// (3) per-StepNo aggregate (find-or-allocate; fixed array, Core §8.11.4(e))
slot := 0;
FOR i := 1 TO PL_Fraktal.MAX_PROFILE_STEPS DO
    IF (StepStats[i].Count > 0) AND (StepStats[i].Id = _openNo) THEN
        slot := i;
        EXIT;
    ELSIF (slot = 0) AND (StepStats[i].Count = 0) THEN
        slot := i;
    END_IF
END_FOR
IF slot = 0 THEN
    StatsTruncated := TRUE;
ELSE
    StepStats[slot].Id    := _openNo;
    StepStats[slot].Label := _openName;
    StepStats[slot].Class := _openClass;
    F_TimingUpdate(Row := StepStats[slot], DurMs := dur);
END_IF
END_METHOD

END_FUNCTION_BLOCK

// ---- BaseClasses/FB_CompositeModuleBase.TcPOU
// Core §2.2 / §8.2 — CM lifecycle + child registry + first-out rollup.
// An EM type registers its children in Setup (_M_Register), ticks them every scan
// (_M_TickChildren, so status stays live whether or not a command runs — Annex B),
// and adopts the first faulted child's diagnostic verbatim (_M_RollupFault).
{attribute 'OPC.UA.DA' := '1'}
FUNCTION_BLOCK ABSTRACT FB_CompositeModuleBase EXTENDS FB_ModuleBase
VAR
    _children : ARRAY[1..PL_Fraktal.MAX_EM_CHILDREN] OF I_Module;
    _nChild   : INT;
END_VAR

Cyclic();

// called from the type's Setup (Core §3.11); bounds-checked per Core §5.6
METHOD PROTECTED _M_Register : BOOL
VAR_INPUT
    Child : I_Module;
END_VAR
IF (Child = 0) OR (_nChild >= PL_Fraktal.MAX_EM_CHILDREN) THEN
    _M_Register := FALSE;
    RETURN;
END_IF
_nChild := _nChild + 1;
_children[_nChild] := Child;
_M_Register := TRUE;
END_METHOD

METHOD PrepareRecipe : BOOL
VAR_INPUT
    Model : ST_ModelId;
END_VAR
VAR
    i, j : INT;
END_VAR
PrepareRecipe := TRUE;
FOR i := 1 TO _nChild DO
    IF (_children[i] <> 0) AND_THEN NOT _children[i].PrepareRecipe(Model := Model) THEN
        PrepareRecipe := FALSE;
        FOR j := 1 TO i DO
            IF _children[j] <> 0 THEN _children[j].AbortRecipe(); END_IF
        END_FOR
        RETURN;
    END_IF
END_FOR
END_METHOD

METHOD CommitRecipe
VAR
    i : INT;
END_VAR
FOR i := 1 TO _nChild DO
    IF _children[i] <> 0 THEN _children[i].CommitRecipe(); END_IF
END_FOR
END_METHOD

METHOD AbortRecipe
VAR
    i : INT;
END_VAR
FOR i := 1 TO _nChild DO
    IF _children[i] <> 0 THEN _children[i].AbortRecipe(); END_IF
END_FOR
END_METHOD

// Core §8.2 — adopt the FIRST faulted child's first-out (reason + child SourcePath)
METHOD PROTECTED _M_RollupFault : BOOL
VAR
    i : INT;
END_VAR
_M_RollupFault := FALSE;
FOR i := 1 TO _nChild DO
    IF _children[i] <> 0 AND_THEN _children[i].FaultActive THEN
        _M_FaultDiag(_children[i].GetFaultSummary());
        _M_RollupFault := TRUE;
        RETURN;
    END_IF
END_FOR
END_METHOD

// children always tick so their status stays live (Annex B §B.3)
METHOD PROTECTED _M_TickChildren
VAR
    i : INT;
END_VAR
FOR i := 1 TO _nChild DO
    IF _children[i] <> 0 THEN
        _children[i].Cyclic();
    END_IF
END_FOR
END_METHOD

PROPERTY ModuleType : E_ModuleType
GET
ModuleType := E_ModuleType.NONE;
END_GET
END_PROPERTY

END_FUNCTION_BLOCK

// ---- BaseClasses/FB_EquipmentModuleBase.TcPOU
// Core §2.2 — discrete-command composite tier. Child recursion lives in
// FB_CompositeModuleBase; this type supplies Equipment Module identity/capability.
FUNCTION_BLOCK ABSTRACT FB_EquipmentModuleBase EXTENDS FB_CompositeModuleBase IMPLEMENTS I_EquipmentModule

PROPERTY ModuleType : E_ModuleType
GET
ModuleType := E_ModuleType.EQUIPMENT_MODULE;
END_GET
END_PROPERTY

END_FUNCTION_BLOCK

// ---- BaseClasses/FB_SequenceBase.TcPOU
// Core §6.8 — THE provided step-chain base: an SFC/ST/LD sequence POU extends
// this and gets the step record, condition waits, run-style pacing, the child
// PLCopen drive, delays, and the shared transition result — without re-declaring
// host plumbing per chain. The derived chart's actions are the only writers of
// _retVal; every chart transition reads it; one shared exit action calls
// M_ClearTransition. Framework flow-control lives here ONCE (§6.8(a)); the
// application's command/wait/decision logic stays visible in each step action.
FUNCTION_BLOCK ABSTRACT FB_SequenceBase
VAR_OUTPUT
    ActiveStep : INT;              // §6.5 mirror of the step record (chart-local view)
    Done : BOOL;                   // finite chains: TRUE at their finish step
END_VAR
VAR
    _step    : INT;                // §6.5 active step index (the ST `CASE _step OF` token)
    _retVal  : E_StepResult;       // shared transition result (§6.10; committed then cleared)
    _restart : BOOL;               // a step may request a chart restart (M_Run applies it)
    {attribute 'OPC.UA.DA' := '0'}
    _host : I_SequenceHost;        // owning module's framework services (§6.7)
    _attached : BOOL;
    _delay : TON;                  // M_Delay's timer (cleared with the transition)
    _driveIssued : BOOL;           // M_MayIssue's per-step issue latch (cleared on commit)
END_VAR

;

// bind the owner's host bridge; the derived Setup adds its typed child bindings.
METHOD M_Attach : BOOL
VAR_INPUT
    Host : I_SequenceHost;
END_VAR
_host := Host;
_attached := (Host <> 0);
M_Attach := _attached;
END_METHOD

// clear the base flow state to the first step. The derived M_Reset calls this.
METHOD M_ResetBase
VAR_INPUT
    FirstStep : INT := 0;          // the chain's initial step number (default N000)
END_VAR
_step := FirstStep;
ActiveStep := FirstStep;
Done := FALSE;
_restart := FALSE;
M_ClearTransition();
END_METHOD

// §6.8 ST-skeleton progression: at the END of a `CASE _step OF` body, commit the
// step's shared transition result. On ADVANCE (or a declared JUMPn) go to the
// mapped next step and clear the step-scoped latches so the new step re-arms — the
// exact guarantee the SFC exit action gave, in one call. NONE stays put. The caller
// passes its successor map; an unmapped result holds the step (safe, visible).
METHOD M_Advance
VAR_INPUT
    OnAdvance : INT;               // next step for E_StepResult.ADVANCE
    OnJump1   : INT := -1;         // next step for JUMP1 (-1 = not used here)
    OnJump2   : INT := -1;
    OnJump3   : INT := -1;
END_VAR
VAR
    target : INT;
END_VAR
target := -1;
CASE _retVal OF
    E_StepResult.ADVANCE: target := OnAdvance;
    E_StepResult.JUMP1:   target := OnJump1;
    E_StepResult.JUMP2:   target := OnJump2;
    E_StepResult.JUMP3:   target := OnJump3;
END_CASE
IF target >= 0 THEN
    _step := target;
    ActiveStep := target;
    M_ClearTransition();           // §6.10: a completed result never leaks into the next step
END_IF
END_METHOD

// the ONE shared exit action: a completed step's result never leaks into the
// next step, and the step-scoped helpers (delay, drive latch) re-arm.
METHOD M_ClearTransition
_retVal := E_StepResult.NONE;
_driveIssued := FALSE;
_delay(IN := FALSE);
END_METHOD

// §6.5 step record + the chart-local ActiveStep mirror, one call.
METHOD M_Step
VAR_INPUT
    StepNo : INT;
    StepName : STRING(120);
    Awaits : I_Module;
    AwaitingLabel : STRING(120);
    Class : E_TimeClass;
    ExpectedTime : TIME;
END_VAR
ActiveStep := StepNo;
IF _host <> 0 THEN
    _host.M_SequenceSetStep(StepNo := StepNo, StepName := StepName, Awaits := Awaits,
        AwaitingLabel := AwaitingLabel, Class := Class, ExpectedTime := ExpectedTime);
END_IF
END_METHOD

// §6.9(b) named plain-condition wait (forward to the host).
METHOD M_Await : BOOL
VAR_INPUT
    Idx : INT;
    Label : STRING(120);
    Ok : BOOL;
END_VAR
M_Await := FALSE;
IF _host <> 0 THEN
    M_Await := _host.M_SequenceAwait(Idx := Idx, Label := Label, Ok := Ok);
END_IF
END_METHOD

// §3.4.2 run-style pacing gate (forward to the host).
METHOD M_Gate : BOOL
VAR_INPUT
    Steppable : BOOL;
END_VAR
M_Gate := FALSE;
IF _host <> 0 THEN
    M_Gate := _host.M_SequenceStepGate(Steppable := Steppable);
END_IF
END_METHOD

// §6.1 issue+await in ONE step: TRUE exactly once per step visit, when the
// run-style gate permits (§3.4.2). The action then sets the child's typed
// Command and raises Execute — visibly, in the step (§6.8). The child's Done
// releases the handshake and sets _retVal := ADVANCE; a child Error needs no
// step code — the owning Unit adopts it instantly via the §8.2 rollup.
// The latch re-arms through the shared exit action (M_ClearTransition).
METHOD M_MayIssue : BOOL
VAR_INPUT
    Steppable : BOOL;
END_VAR
M_MayIssue := FALSE;
IF _driveIssued THEN
    RETURN;
END_IF
IF M_Gate(Steppable := Steppable) THEN
    _driveIssued := TRUE;
    M_MayIssue := TRUE;
END_IF
END_METHOD

// a declared process wait in ONE step (settle/dwell). The timer runs while the
// step is active and re-arms through the shared exit action.
METHOD M_Delay : E_StepResult
VAR_INPUT
    PT : TIME;
END_VAR
M_Delay := E_StepResult.NONE;
_delay(IN := TRUE, PT := PT);
IF _delay.Q THEN
    _delay(IN := FALSE);
    M_Delay := E_StepResult.ADVANCE;
END_IF
END_METHOD

// §3.16.3 forward (framework plumbing stays out of step actions).
METHOD M_PartReceived : BOOL
M_PartReceived := FALSE;
IF _host <> 0 THEN
    M_PartReceived := _host.M_SequencePartReceived();
END_IF
END_METHOD

METHOD M_PartStarted
IF _host <> 0 THEN
    _host.M_SequencePartStarted();
END_IF
END_METHOD

METHOD M_PartRecord : BOOL
VAR_INPUT
    RecordName : STRING(64);
    Value : LREAL;
    Minimum : LREAL;
    Maximum : LREAL;
    Target : LREAL;
    EngUnit : STRING(16);
END_VAR
M_PartRecord := FALSE;
IF _host <> 0 THEN
    M_PartRecord := _host.M_SequencePartRecord(RecordName := RecordName,
        Value := Value, Minimum := Minimum, Maximum := Maximum, Target := Target,
        EngUnit := EngUnit);
END_IF
END_METHOD

METHOD M_PartProcessed : BOOL
VAR_INPUT
    Verdict : E_Verdict;
    Reason : E_Reason;
END_VAR
M_PartProcessed := FALSE;
IF _host <> 0 THEN
    M_PartProcessed := _host.M_SequencePartProcessed(Verdict := Verdict, Reason := Reason);
END_IF
END_METHOD

METHOD M_CountGood
IF _host <> 0 THEN
    _host.M_SequenceCountGood();
END_IF
END_METHOD

// §6.11 forward
METHOD M_AskDecision
VAR_INPUT
    Req : ST_DecisionRequest;
END_VAR
IF _host <> 0 THEN
    _host.M_SequenceAskDecision(Req := Req);
END_IF
END_METHOD

METHOD M_TakeDecision : INT
M_TakeDecision := 0;
IF _host <> 0 THEN
    M_TakeDecision := _host.M_SequenceTakeDecision();
END_IF
END_METHOD

METHOD M_ClearDecision
IF _host <> 0 THEN
    _host.M_SequenceClearDecision();
END_IF
END_METHOD

// §6.1 one-shot completion forward (finite chains)
METHOD M_Complete
IF _host <> 0 THEN
    _host.M_SequenceComplete();
END_IF
END_METHOD

// §8.11.1 cycle-complete marker forward; FALSE = stop granted (do not loop)
METHOD M_EndOfCycle : BOOL
M_EndOfCycle := FALSE;
IF _host <> 0 THEN
    M_EndOfCycle := _host.M_SequenceEndOfCycle();
END_IF
END_METHOD

// §3.4 — poll at the between-cycles wait step (forward to the host).
METHOD M_StopPending : BOOL
M_StopPending := FALSE;
IF _host <> 0 THEN
    M_StopPending := _host.M_SequenceStopPending();
END_IF
END_METHOD

// §3.4/§8.11 — accept the stop between cycles (forward to the host).
METHOD M_StopNow
IF _host <> 0 THEN
    _host.M_SequenceStopNow();
END_IF
END_METHOD

// §6.9 first-out fault from a step (forward to the host).
METHOD M_Fault
VAR_INPUT
    Reason : E_Reason;
    DescriptionKey : STRING(255);
END_VAR
IF _host <> 0 THEN
    _host.M_SequenceFault(Reason := Reason, DescriptionKey := DescriptionKey);
END_IF
END_METHOD

END_FUNCTION_BLOCK

// ---- BaseClasses/FB_UnitBase.TcPOU
// Core §2.2 lifecycle family, top tier: modes + cascade (§3.4/§3.7), Start/Stop
// mapped onto the §6.1 run command (§6 intro), the step chain (_M_SetStep/_M_Await,
// §6.5/§6.9(b)), the stall walk as a PENDING reason with instant rollup on an
// awaited module's Error (§6.9/§8.2), the §8.11.4 profiler wired in, and
// Starved/Blocked derived from the step's time class (§8.11.4(f)/§8.11.3).
// A Unit type overrides _M_Dispatch (its mode chain) + _M_Supports (+ §3.14 hooks).
{attribute 'OPC.UA.DA' := '1'}
FUNCTION_BLOCK ABSTRACT FB_UnitBase EXTENDS FB_CompositeModuleBase IMPLEMENTS I_Unit, I_SequenceHost
VAR_INPUT
    DecisionAnswer : INT;              // §6.11: chosen option index (0 = none yet)
    ReqControlOn   : BOOL;             // §9.8 HMI/data request; edge-consumed and access-gated
    ReqControlOff  : BOOL;
    HmiRequest     : ST_HmiRequest;     // §3.10/§14: arguments first, Sequence last
    {attribute 'OPC.UA.DA' := '0'}
    ControlDomain  : ST_ControlDomainStatus; // §9.8: optional shared cell/cage arrangement
END_VAR
VAR_OUTPUT
    Starved : BOOL;                    // §8.11.3 — derived from CurrentStep.Class
    Blocked : BOOL;
    Domain  : ST_ControlDomainStatus;  // §9.8 read-only publication of the assigned domain
    ControlOnRequest  : BOOL;          // one-scan request to the owning domain coordinator
    ControlOffRequest : BOOL;
END_VAR
VAR_OUTPUT
    Profiler    : FB_CycleProfiler;    // §8.11.4 — HMI chart source
    CurrentStep : ST_StepRecord;       // §6.5 — feeds §6.9 walk AND the profiler
    Pending     : ST_Diagnostic;       // live stall reason (Low) — NOT a fault (§6.9)
    Decision    : ST_DecisionRequest;  // §6.11 active request ('' Prompt = none)
    StallTime   : TIME := T#30S;       // guard when the step declares no ExpectedTime
    Model       : ST_ModelId;          // §3.1b active model identity (published for HMI/MES/trace)
    AvailableModelCount : INT;         // §3.8 optional discoverable model/recipe catalog
    AvailableModels : ARRAY[1..PL_Fraktal.MAX_RECIPES] OF ST_ModelId;
    Part        : ST_PartContext;      // §3.16.1 live part context (Present=FALSE, Uid='' = none)
    AlarmLog    : FB_AlarmLog;         // §8.3 — active list + closed ring + Blocking
    Access      : FB_AccessManager;    // §7.7 — per-root session/policy (default: fully open)
    GoodCount   : UDINT;               // §8.11.2 — cycle verdict counters
    NokCount    : UDINT;
    ReworkCount : UDINT;
    NokReason   : E_Reason;            // §8.11.2 — last NOK's first-out attribution
    MachineState : E_MachineState;     // §8.11.3 — classified every scan (OEE/PackML/host)
    History     : ARRAY[1..PL_Fraktal.MAX_DIAG_RING] OF ST_Diagnostic;  // §6.9(a) ring (newest at HistoryHead)
    HistoryHead : INT;
    ModePolicy  : ARRAY[0..PL_Fraktal.MODE_COUNT-1] OF ST_ModePolicy;    // §3.4.1 per-mode switch policy (station cfg)
    RunStyle    : E_RunStyle;          // §3.4.2 active run style (HMI-selectable; CONTINUOUS default)
    Oee         : ST_Oee;              // §8.5.1 accumulators + snapshot (published)
    OeeTrend    : ARRAY[1..PL_Fraktal.MAX_OEE_SAMPLES] OF ST_OeeSample; // §8.5.1 ring
    OeeTrendHead: INT;                 // newest sample index (0 = none yet)
    HmiResponse : ST_HmiResponse;
    ModeActivePublished : E_Mode;       // properties are not OPC UA-visible
    RunningPublished : BOOL;
    StopPendingPublished : BOOL;
    SupportedModesPublished : ARRAY[0..PL_Fraktal.MODE_COUNT-1] OF BOOL;
    SupportedRunStylesPublished : ARRAY[0..2] OF BOOL;
END_VAR
VAR
    _fTrig    : R_TRIG;
    _mode     : E_Mode;
    _modeReq  : E_Mode;
    _modePend : BOOL;
    _stopReq  : BOOL;
    _awaits   : I_Module;              // module the current step awaits (0 = none)
    _faultEvt : INT;                   // open ERROR event slot in AlarmLog (0 = none)
    _tStall   : TON;
    _stepReq  : BOOL;                  // §3.4.2 pending single-step request (edge-consumed)
    _holdRun  : BOOL;                  // §3.4.2 HOLD_TO_RUN input held (NON-SAFETY, §9)
    _stepArm  : R_TRIG;
    _oeeLast  : TIME;                  // §8.5.1 last accumulation stamp
    _oeeSampMs: UDINT;                 // ms since last trend sample
    _hmiLastSequence : UDINT;
    _carrier  : I_PartCarrier;         // §3.16.2 injected part carrier (0 = traceability off)
END_VAR

Cyclic();

// base first (§3.14.2); then children, one-shot init, mode transition, stall watch
METHOD PROTECTED OnCyclic : DINT
VAR
    publishIdx : INT;
    modeIdx    : E_Mode;
    styleIdx   : E_RunStyle;
END_VAR
OnCyclic := SUPER^.OnCyclic();
_M_TickChildren();
_M_OeeUpdate();                                       // §8.5.1 time accounting + sampling
AlarmLog.Cyclic();                                    // §8.10 shelf auto-expiry
_M_HandleHmiRequest();                                // §3.10 request mailbox
Access.Cyclic();
// §9.8 data-driven Control On/Off request endpoint. Off wins if both arrive;
// the domain/power-group implementation still validates safety, health and rearm.
ControlOnRequest := FALSE;
ControlOffRequest := FALSE;
IF ReqControlOff THEN
    ReqControlOff := FALSE;
    ReqControlOn := FALSE;
    IF Access.PermitsLogged(Gate := E_GatedAction.POWER_CONTROL) THEN
        ControlOffRequest := TRUE;
    END_IF
ELSIF ReqControlOn THEN
    ReqControlOn := FALSE;
    IF Access.PermitsLogged(Gate := E_GatedAction.POWER_CONTROL) THEN
        ControlOnRequest := TRUE;
    END_IF
END_IF
// §3.14.4 — pending mode change; §3.4.1 style decides graceful vs immediate
IF _modePend THEN
    IF _exec = E_ExecState.BUSY THEN
        IF ModePolicy[TO_INT(_mode)].Style = E_ModeSwitchStyle.GRACEFUL THEN
            _stopReq := TRUE;                             // finish the cycle at its stop point
        ELSIF OnModeExit() = 0 THEN
            OnAbort();                                    // IMMEDIATE: cancel now (override may defer)
        END_IF
    ELSE
        IF _exec <> E_ExecState.READY THEN
            Execute := FALSE;                             // release the run command (§6.1 reset)
        ELSE
            _mode := _modeReq;
            _modePend := FALSE;
            _M_CascadeMode(_mode);                        // §3.7 cascade [TC3]
            OnModeChanged();
        END_IF
    END_IF
END_IF
// §8.3(c) — automatic fault capture: ERROR entry raises, ERROR exit marks gone
IF (_exec = E_ExecState.ERROR) AND (_faultEvt = 0) THEN
    _faultEvt := AlarmLog.RaiseDiag(D := _diag, ResetClass := E_ResetClass.MANUAL_RESET);
    _M_PartAborted();                  // §3.16.3: a faulted part leaves without a valid result
ELSIF (_exec <> E_ExecState.ERROR) AND (_faultEvt > 0) THEN
    AlarmLog.Gone(Slot := _faultEvt);                            // -> WAIT_RESET (blocking)
    _faultEvt := 0;
END_IF
// §6.9 — instant rollup on awaited Error; stall as PENDING otherwise
IF _exec = E_ExecState.BUSY THEN
    IF (_awaits <> 0) AND_THEN _awaits.FaultActive THEN
        _M_FaultDiag(_awaits.GetFaultSummary());
    ELSE
        _tStall(IN := TRUE, PT := SEL(CurrentStep.ExpectedTime > T#0S, StallTime, CurrentStep.ExpectedTime));
        IF _tStall.Q THEN
            _M_StallWalk();
        END_IF
    END_IF
ELSE
    _tStall(IN := FALSE);
END_IF
// §6.9(a) — every new fault joins the shift-change ring, no historian needed
_fTrig(CLK := (_exec = E_ExecState.ERROR));
IF _fTrig.Q THEN
    _M_PushHistory(_diag);
END_IF
// §8.11.4(d) — creeping WORK time is a MAINTENANCE event (Low), not downtime:
// the profiler pulses once per excursion past the configured baseline band.
IF Profiler.DegradedTrig THEN
    _M_RaiseMaintenance(Reason := E_Reason.CYCLE_TIME_DEGRADED,
        Text := 'std.maintenance.cycleTimeDegraded');
END_IF
ModeActivePublished := _mode;
RunningPublished := (_exec = E_ExecState.BUSY);
StopPendingPublished := _stopReq AND (_exec = E_ExecState.BUSY);
FOR publishIdx := 0 TO PL_Fraktal.MODE_COUNT - 1 DO
    modeIdx := publishIdx;
    SupportedModesPublished[publishIdx] := _M_Supports(Mode := modeIdx);
END_FOR
FOR publishIdx := 0 TO 2 DO
    styleIdx := publishIdx;
    SupportedRunStylesPublished[publishIdx] := _M_SupportsRunStyle(Style := styleIdx);
END_FOR
END_METHOD

// §3.14 hook — one-shot after first operational scan
METHOD PROTECTED OnInit : DINT
OnInit := SUPER^.OnInit();
Access.Setup(Provider := 0, pAlarmLog := ADR(AlarmLog)); // preserves an injected provider
_M_InitModePolicy();
END_METHOD

// §6.9/§3.10(a') — overlay the pending stall after the common mirror refresh.
METHOD PROTECTED _M_PublishStatus
SUPER^._M_PublishStatus();
// §8.11.4(f)/§8.11.3 — one declaration, two views. Derived AFTER dispatch so the
// wait class reflects the step record this scan just set, not the previous one.
Starved := (_exec = E_ExecState.BUSY) AND (CurrentStep.Class = E_TimeClass.WAIT_UPSTREAM);
Blocked := (_exec = E_ExecState.BUSY) AND (CurrentStep.Class = E_TimeClass.WAIT_DOWNSTREAM);
// §8.11.3 — classify into the fixed machine-state set (priority: fault first,
// then planned states, then line attribution, then producing/idle).
IF (_exec = E_ExecState.ERROR) OR AlarmLog.Blocking THEN
    MachineState := E_MachineState.DOWN;
ELSIF _mode = E_Mode.CHANGEOVER THEN
    MachineState := E_MachineState.CHANGEOVER;
ELSIF Blocked THEN
    MachineState := E_MachineState.BLOCKED;
ELSIF Starved THEN
    MachineState := E_MachineState.STARVED;
ELSIF _exec = E_ExecState.BUSY THEN
    MachineState := E_MachineState.PRODUCING;
ELSIF _stopReq OR (_exec = E_ExecState.ABORTED) THEN
    MachineState := E_MachineState.STOPPED;
ELSE
    MachineState := E_MachineState.IDLE;
END_IF
Status.ControlDomainId := ControlDomain.Id;
Domain := ControlDomain;
Safety := ControlDomain.Safety;             // read-only HMI mirror; ownership stays in domain
ControlPower := ControlDomain.ControlPower;
IF (_exec <> E_ExecState.ERROR) AND (Pending.ReasonCode <> E_Reason.NONE) THEN
    Status.Diagnostic := Pending;
END_IF
END_METHOD

// §8.11.4(d)/§8.12 — a Low-severity maintenance event: informs planning, does not
// stop the cycle. Instant come+gone ring entry (the trend data lives in Profiler).
METHOD PROTECTED _M_RaiseMaintenance
VAR_INPUT
    Reason : E_Reason;
    Text : STRING(255);
END_VAR
VAR
    slot : INT;
END_VAR
slot := AlarmLog.Raise(Reason := Reason, Text := Text, Source := _name,
    Severity := E_Severity.LOW, Category := E_Category.SYSTEM,
    ResetClass := E_ResetClass.AUTO_RESET);
IF slot > 0 THEN
    AlarmLog.Gone(Slot := slot);
END_IF
END_METHOD

// I_SequenceHost (§6.7/§6.8) — step record for a separately-compiled chain.
METHOD M_SequenceSetStep
VAR_INPUT
    StepNo : INT;
    StepName : STRING(120);
    Awaits : I_Module;
    AwaitingLabel : STRING(120);
    Class : E_TimeClass;
    ExpectedTime : TIME;
END_VAR
_M_SetStep(StepNo := StepNo, StepName := StepName,
    Awaits := Awaits, AwaitingLabel := AwaitingLabel, Class := Class,
    ExpectedTime := ExpectedTime);
END_METHOD

METHOD M_SequenceAwait : BOOL
VAR_INPUT
    Idx : INT;
    Label : STRING(120);
    Ok : BOOL;
END_VAR
M_SequenceAwait := _M_Await(Idx := Idx, Label := Label, Ok := Ok);
END_METHOD

METHOD M_SequenceStepGate : BOOL
VAR_INPUT
    Steppable : BOOL;
END_VAR
M_SequenceStepGate := _M_StepGate(Steppable := Steppable);
END_METHOD

METHOD M_SequencePartReceived : BOOL
M_SequencePartReceived := _M_PartReceived();
END_METHOD

METHOD M_SequencePartStarted
_M_PartStarted();
END_METHOD

METHOD M_SequencePartRecord : BOOL
VAR_INPUT
    RecordName : STRING(64);
    Value : LREAL;
    Minimum : LREAL;
    Maximum : LREAL;
    Target : LREAL;
    EngUnit : STRING(16);
END_VAR
M_SequencePartRecord := _M_PartRecord(RecordName := RecordName,
    Value := Value, Minimum := Minimum, Maximum := Maximum, Target := Target,
    EngUnit := EngUnit);
END_METHOD

METHOD M_SequencePartProcessed : BOOL
VAR_INPUT
    Verdict : E_Verdict;
    Reason : E_Reason;
END_VAR
M_SequencePartProcessed :=
    _M_PartProcessed(Verdict := Verdict, Reason := Reason);
END_METHOD

METHOD M_SequenceCountGood
CountGood();
END_METHOD

METHOD M_SequenceAskDecision
VAR_INPUT
    Req : ST_DecisionRequest;
END_VAR
_M_AskDecision(Req := Req);
END_METHOD

METHOD M_SequenceTakeDecision : INT
M_SequenceTakeDecision := _M_TakeDecision();
END_METHOD

METHOD M_SequenceClearDecision
Decision.Prompt := '';
DecisionAnswer := 0;
END_METHOD

METHOD M_SequenceComplete
_M_Complete();
END_METHOD

METHOD M_SequenceEndOfCycle : BOOL
M_SequenceEndOfCycle := _M_EndOfCycle();
END_METHOD

METHOD M_SequenceFault
VAR_INPUT
    Reason : E_Reason;
    DescriptionKey : STRING(255);
END_VAR
_M_Fault(Reason, DescriptionKey);
END_METHOD

// §3.4 — a chain polls this at its between-cycles wait step.
METHOD M_SequenceStopPending : BOOL
M_SequenceStopPending := _stopReq AND (_exec = E_ExecState.BUSY);
END_METHOD

// §3.4/§8.11 — accept a pending Stop BETWEEN cycles: the open profile fragment
// (just the wait step) is abandoned, not published as a production cycle.
METHOD M_SequenceStopNow
Profiler.CycleAbandon();
_stopReq := FALSE;
Execute := FALSE;
_M_Complete();
END_METHOD

// §3.16.2 — inject the part carrier at the composition root (0 = traceability off).
// Source-agnostic: BY_POSITION local, RFID, DataMatrix, or host, behind I_PartCarrier.
METHOD SetPartCarrier : BOOL
VAR_INPUT
    Carrier : I_PartCarrier;
END_VAR
_carrier := Carrier;
SetPartCarrier := (Carrier <> 0);
END_METHOD

// §3.16.3 — one canonical part-lifecycle event: instant come+gone MESSAGE ring entry.
METHOD PRIVATE _M_PartEvent
VAR_INPUT
    Reason : E_Reason;
    Text : STRING(255);
END_VAR
VAR
    slot : INT;
    txt : STRING(255);
END_VAR
txt := CONCAT(Text, Part.Uid);
slot := AlarmLog.Raise(Reason := Reason, Text := txt, Source := _name,
    Severity := E_Severity.LOW, Category := E_Category.PROCESS,
    ResetClass := E_ResetClass.AUTO_RESET);
IF slot > 0 THEN
    AlarmLog.Gone(Slot := slot);
END_IF
END_METHOD

// §3.16.3 EVENT_PART_RECEIVED — confirm identity at station entry via the carrier.
// FALSE with a CARRIER_READ_FAILED fault on a failed read (never silent), FALSE
// silently when no carrier is configured (§3.9 feature selectability).
METHOD PROTECTED _M_PartReceived : BOOL
VAR
    i : INT;
END_VAR
_M_PartReceived := FALSE;
IF _carrier = 0 THEN
    RETURN;
END_IF
Part.Uid := '';                              // station entry = fresh identity read
IF NOT _carrier.ReadContext(Ctx := Part) THEN
    _M_Fault(E_Reason.CARRIER_READ_FAILED, 'std.error.partCarrierReadFailed');
    RETURN;
END_IF
Part.Result.Verdict := E_Verdict.NONE;       // this station's outcome starts empty
Part.Result.ReasonCode := E_Reason.NONE;
Part.Result.StationPath := _name;
FOR i := 1 TO PL_Fraktal.MAX_RESULTS DO
    Part.Result.Records[i].Name := '';
END_FOR
_M_PartEvent(Reason := E_Reason.EVENT_PART_RECEIVED, Text := 'std.event.partReceived: ');
_M_PartReceived := TRUE;
END_METHOD

// §3.16.3 EVENT_PART_PROCESSING_STARTED — the value-adding sequence begins.
METHOD PROTECTED _M_PartStarted
IF (_carrier = 0) OR NOT Part.Present THEN
    RETURN;
END_IF
_M_PartEvent(Reason := E_Reason.EVENT_PART_PROCESSING_STARTED,
    Text := 'std.event.partProcessingStarted: ');
END_METHOD

// §3.16.1 — append one measured value to this part's result (test cells).
// FALSE when the bounded record table is full (RESULT_RECORD_REJECTED semantics).
METHOD PROTECTED _M_PartRecord : BOOL
VAR_INPUT
    RecordName : STRING(64);
    Value : LREAL;
    Minimum : LREAL;
    Maximum : LREAL;
    Target : LREAL;
    EngUnit : STRING(16);
END_VAR
VAR
    i : INT;
END_VAR
_M_PartRecord := FALSE;
IF NOT Part.Present THEN
    RETURN;
END_IF
FOR i := 1 TO PL_Fraktal.MAX_RESULTS DO
    IF Part.Result.Records[i].Name = '' THEN
        Part.Result.Records[i].Name := RecordName;
        Part.Result.Records[i].Value := Value;
        Part.Result.Records[i].Minimum := Minimum;
        Part.Result.Records[i].Maximum := Maximum;
        Part.Result.Records[i].Target := Target;
        Part.Result.Records[i].Unit := EngUnit;
        Part.Result.Records[i].InTol := (Maximum <= Minimum)
            OR ((Value >= Minimum) AND (Value <= Maximum));
        _M_PartRecord := TRUE;
        RETURN;
    END_IF
END_FOR
END_METHOD

// §3.16.3 EVENT_PART_PROCESSED — stamp the verdict, write the carrier FIRST
// (result-before-event contract), then raise the event. The Uid and result stay
// published until the next part so the HMI shows the last outcome.
METHOD PROTECTED _M_PartProcessed : BOOL
VAR_INPUT
    Verdict : E_Verdict;
    Reason : E_Reason;
END_VAR
_M_PartProcessed := FALSE;
IF (_carrier = 0) OR NOT Part.Present THEN
    RETURN;
END_IF
Part.Result.Verdict := Verdict;
Part.Result.ReasonCode := Reason;
Part.Result.StationPath := _name;
Part.Result.Stamp := F_Now();
IF NOT _carrier.WriteResult(Ctx := Part) THEN
    _M_Fault(E_Reason.CARRIER_WRITE_FAILED, 'std.error.partCarrierWriteFailed');
    RETURN;
END_IF
// §8.11.2 — counters increment HERE, from the verdict; an NOK carries its
// first-out ReasonCode so scrap is analysable by cause (§8.8 vocabulary).
CASE Verdict OF
    E_Verdict.OK:     CountGood();
    E_Verdict.NOK:    CountNok();    NokReason := Reason;
    E_Verdict.REWORK: CountRework();
ELSE
    ;                                // NONE: no count — the part left unjudged
END_CASE
_M_PartEvent(Reason := E_Reason.EVENT_PART_PROCESSED, Text := 'std.event.partProcessed: ');
Part.Present := FALSE;
_M_PartProcessed := TRUE;
END_METHOD

// §3.16.3 EVENT_PART_PROCESSING_ABORTED — the part leaves without a valid result
// (fault, abort, manual removal). Called automatically on Unit ERROR entry.
METHOD PROTECTED _M_PartAborted
IF (_carrier = 0) OR NOT Part.Present THEN
    RETURN;
END_IF
Part.Result.Verdict := E_Verdict.NONE;
_M_PartEvent(Reason := E_Reason.EVENT_PART_PROCESSING_ABORTED,
    Text := 'std.event.partAborted: ');
Part.Present := FALSE;
END_METHOD

// §3.14 hook — after the new mode is committed
METHOD PROTECTED OnModeChanged : DINT
OnModeChanged := 0;
END_METHOD

// §3.14.4 — called every scan while a mode request is pending and the Unit is BUSY.
// Return 0 = consent to immediate cancel (default); >0 = still stopping gracefully.
METHOD PROTECTED OnModeExit : DINT
OnModeExit := 0;
END_METHOD

// §3.4/§3.7 — FALSE = unsupported (graceful rejection); TRUE = committed or pending
METHOD SetMode : BOOL
VAR_INPUT
    Mode : E_Mode;
END_VAR
IF NOT Access.PermitsLogged(Gate := E_GatedAction.MODE_CHANGE) THEN
    SetMode := FALSE;                  // §7.7(c): who-gate ANDs the machine gates
    RETURN;
END_IF
IF NOT _M_Supports(Mode) THEN
    SetMode := FALSE;
    RETURN;
END_IF
IF (Mode = _mode) AND NOT _modePend THEN
    SetMode := TRUE;
    RETURN;
END_IF
// §3.4.1 shield: policy of the mode being LEFT governs while its sequence runs
IF (_exec = E_ExecState.BUSY)
AND (ModePolicy[TO_INT(_mode)].Shield = E_ModeSwitchShield.BLOCKED_WHILE_RUNNING) THEN
    SetMode := FALSE;                  // must Stop first (graceful rejection, not a fault)
    RETURN;
END_IF
_modeReq := Mode;
_modePend := TRUE;
SetMode := TRUE;
END_METHOD

// §3.3/§6 intro — the run IS a §6.1 command.
// §7.8: ReleaseReportStart is the authoritative machine gate as well as the
// operator explanation, so a concrete Unit cannot report an interlock it ignores.
// Build directly into the published response storage: ST_ReleaseReport is too
// large for nested by-value/local copies on a small TwinCAT task stack.
METHOD Start : BOOL
IF NOT Access.PermitsLogged(Gate := E_GatedAction.START_STOP) THEN
    Start := FALSE;                    // §7.7
    RETURN;
END_IF
IF ReleaseReportStart(Report := HmiResponse.Report) THEN
    _stopReq := FALSE;                 // §8.3(b): a MANUAL_RESET event blocks restart
    Execute := TRUE;
    Start := TRUE;
ELSE
    Start := FALSE;
END_IF
END_METHOD

// §3.3 — stop after the current cycle
METHOD Stop : BOOL
IF NOT Access.PermitsLogged(Gate := E_GatedAction.START_STOP) THEN
    Stop := FALSE;                     // §7.7
    RETURN;
END_IF
IF _exec = E_ExecState.BUSY THEN
    _stopReq := TRUE;
ELSE
    _stopReq := FALSE;
    Execute := FALSE;                  // release a terminal run command (ERROR/DONE/ABORTED)
END_IF
Stop := TRUE;
END_METHOD

// §6.11 — publish a typed decision request (single active slot)
METHOD PROTECTED _M_AskDecision
VAR_INPUT
    Req : ST_DecisionRequest;
END_VAR
Decision := Req;
Decision.SourcePath := _name;
END_METHOD

// §6.9(b) — named plain-condition wait; returns the condition so steps read naturally
METHOD PROTECTED _M_Await : BOOL
VAR_INPUT
    Idx   : INT;
    Label : STRING(120);
    Ok    : BOOL;
END_VAR
IF (Idx >= 1) AND (Idx <= PL_Fraktal.MAX_STEP_CONDS) THEN
    CurrentStep.Conds[Idx].Label := Label;
    CurrentStep.Conds[Idx].Ok    := Ok;
END_IF
_M_Await := Ok;
END_METHOD

// §3.7 — offer the mode to child Units; a child may reject (graceful)
METHOD PROTECTED _M_CascadeMode
VAR_INPUT
    Mode : E_Mode;
END_VAR
VAR
    i  : INT;
    iu : I_Unit;
END_VAR
FOR i := 1 TO _nChild DO
    IF _children[i] <> 0 THEN
        IF __QUERYINTERFACE(_children[i], iu) THEN   // [TC3] capability query — TC3 §3.2
            iu.SetMode(Mode);
        END_IF
    END_IF
END_FOR
END_METHOD

METHOD PROTECTED _M_ClearPending
Pending.ReasonCode  := E_Reason.NONE;
Pending.Description := '';
END_METHOD

// call at the finish step (§8.11.1): publishes the profile; FALSE = stop granted
METHOD PROTECTED _M_EndOfCycle : BOOL
Profiler.CycleComplete();
IF _stopReq THEN
    _stopReq := FALSE;
    Execute := FALSE;
    _M_Complete();
    _M_EndOfCycle := FALSE;
ELSE
    _M_EndOfCycle := TRUE;
END_IF
END_METHOD

// §6.5 — the ONE line per step: record for the §6.9 walk AND the §8.11.4 profiler
METHOD PROTECTED _M_SetStep
VAR_INPUT
    StepNo        : INT;
    StepName      : STRING(120);
    Awaits        : I_Module;
    AwaitingLabel : STRING(120);
    Class         : E_TimeClass;
    ExpectedTime  : TIME;
END_VAR
VAR
    i : INT;
    e : ST_CondRecord;
END_VAR
IF StepNo <> CurrentStep.StepNo THEN
    _tStall(IN := FALSE);
    _M_ClearPending();
    FOR i := 1 TO PL_Fraktal.MAX_STEP_CONDS DO
        CurrentStep.Conds[i] := e;
    END_FOR
END_IF
CurrentStep.StepNo        := StepNo;
CurrentStep.StepName      := StepName;
CurrentStep.AwaitingLabel := AwaitingLabel;
CurrentStep.Class         := Class;
CurrentStep.ExpectedTime  := ExpectedTime;
_awaits := Awaits;
Profiler.StepChanged(StepNo := StepNo, StepName := StepName, Class := Class,
    Expected := ExpectedTime);
END_METHOD

// §6.9 — build the pending stall reason: step -> awaited command -> first FALSE condition
METHOD PROTECTED _M_StallWalk
IF Pending.ReasonCode = E_Reason.NONE THEN
    Pending.Since := F_Now();
END_IF
Pending.ReasonCode := E_Reason.STEP_STALLED;
Pending.Severity   := E_Severity.LOW;
Pending.Category   := E_Category.PROCESS;
Pending.SourcePath := _name;
Pending.Description := 'std.diagnostic.stepStalled';
END_METHOD

// §3.4 — override to declare the type's mode set (baseline: AUTO + MANUAL)
METHOD PROTECTED _M_Supports : BOOL
VAR_INPUT
    Mode : E_Mode;
END_VAR
_M_Supports := (Mode = E_Mode.AUTO) OR (Mode = E_Mode.MANUAL);
END_METHOD

// §6.11 — returns the chosen option once and clears the request (0 = none yet)
METHOD PROTECTED _M_TakeDecision : INT
IF DecisionAnswer > 0 THEN
    _M_TakeDecision := DecisionAnswer;
    DecisionAnswer := 0;
    Decision.Prompt := '';
ELSE
    _M_TakeDecision := 0;
END_IF
END_METHOD

// §8.11 — called by the chain/verdict glue at part completion
METHOD CountGood : BOOL
GoodCount := GoodCount + 1;
CountGood := TRUE;
END_METHOD

// §8.11.2 — REWORK verdict counter (see CountGood)
METHOD CountRework : BOOL
ReworkCount := ReworkCount + 1;
CountRework := TRUE;
END_METHOD

METHOD CountNok : BOOL
NokCount := NokCount + 1;
CountNok := TRUE;
END_METHOD

// §6.9(a) — fixed ring, newest at HistoryHead; never allocates
METHOD PROTECTED _M_PushHistory
VAR_INPUT
    D : ST_Diagnostic;
END_VAR
HistoryHead := (HistoryHead MOD PL_Fraktal.MAX_DIAG_RING) + 1;
History[HistoryHead] := D;
END_METHOD

// §3.1b/§3.8 — transactional model change: prepare the whole subtree, then commit.
METHOD SetModel : BOOL
VAR_INPUT
    Id : ST_ModelId;
END_VAR
IF NOT Access.PermitsLogged(Gate := E_GatedAction.CHANGEOVER) THEN
    SetModel := FALSE;                 // §7.7
    RETURN;
END_IF
IF _exec = E_ExecState.BUSY THEN
    SetModel := FALSE;                 // changeover is not mid-cycle (§3.8 loads at CHANGEOVER)
    RETURN;
END_IF
IF NOT PrepareRecipe(Model := Id) THEN
    AbortRecipe();
    SetModel := FALSE;
    RETURN;
END_IF
CommitRecipe();                         // infallible after successful preparation
Model := Id;                           // identity changes only after subtree commit
SetModel := TRUE;
END_METHOD

// §3.8 optional HMI/MES selection catalog. Recipe providers remain pluggable;
// the application registers only the model identities it deliberately exposes.
METHOD RegisterAvailableModel : BOOL
VAR_INPUT
    Id : ST_ModelId;
END_VAR
VAR
    i : INT;
END_VAR
RegisterAvailableModel := FALSE;
IF (Id.ModelCode = '') OR (AvailableModelCount >= PL_Fraktal.MAX_RECIPES) THEN
    RETURN;
END_IF
FOR i := 1 TO AvailableModelCount DO
    IF AvailableModels[i].ModelCode = Id.ModelCode THEN
        RETURN;
    END_IF
END_FOR
AvailableModelCount := AvailableModelCount + 1;
AvailableModels[AvailableModelCount] := Id;
RegisterAvailableModel := TRUE;
END_METHOD

// §8.3(b) — deliberate operator reset of blocking events (release-gated per §7.6/§14).
// Closes WAIT_RESET events; an event whose condition persists stays ACTIVE.
METHOD OperatorReset : BOOL
IF NOT Access.PermitsLogged(Gate := E_GatedAction.ALARM_RESET) THEN
    OperatorReset := FALSE;            // §7.7
    RETURN;
END_IF
OperatorReset := AlarmLog.OperatorReset();
END_METHOD

PROPERTY ModeActive : E_Mode
GET
ModeActive := _mode;
END_GET
END_PROPERTY

PROPERTY ModelCode : STRING(64)
GET
ModelCode := Model.ModelCode;
END_GET
END_PROPERTY

PROPERTY ModuleType : E_ModuleType
GET
ModuleType := E_ModuleType.UNIT;
END_GET
END_PROPERTY

// §7.6.1 — single gated manual-command entry for the HMI. Accepts ONLY when this
// Unit is in MANUAL (§3.4) AND the user holds MANUAL access (§7.7). Routes to the
// target module's ManualCommand (through the command surface — defended, not
// bypassed). Logs every accept/reject as a §8.3 event. Concrete Units override
// _M_RouteManual to map TargetPath -> the child module.
METHOD ManualCommandTo : BOOL
VAR_INPUT
    TargetPath : STRING(255);
    Value : DINT;
END_VAR
VAR
    auditSlot : INT;
END_VAR
ManualCommandTo := FALSE;
IF _mode <> E_Mode.MANUAL THEN
    auditSlot := AlarmLog.Raise(Reason := E_Reason.NONE,
        Text := 'std.audit.manualCommandWrongMode', Source := TargetPath,
        Severity := E_Severity.LOW, Category := E_Category.SYSTEM, ResetClass := E_ResetClass.AUTO_RESET);
    IF auditSlot > 0 THEN AlarmLog.Gone(Slot := auditSlot); END_IF
    RETURN;
END_IF
IF NOT Access.PermitsLogged(Gate := E_GatedAction.MANUAL) THEN
    RETURN;                              // §7.7 denial already audited
END_IF
ManualCommandTo := _M_RouteManual(TargetPath := TargetPath, Value := Value);
IF ManualCommandTo THEN
    auditSlot := AlarmLog.Raise(Reason := E_Reason.NONE,
        Text := 'std.audit.manualCommandAccepted', Source := TargetPath,
        Severity := E_Severity.LOW, Category := E_Category.SYSTEM, ResetClass := E_ResetClass.AUTO_RESET);
ELSE
    auditSlot := AlarmLog.Raise(Reason := E_Reason.UNSUPPORTED_COMMAND,
        Text := 'std.audit.manualCommandRejected', Source := TargetPath,
        Severity := E_Severity.LOW, Category := E_Category.SYSTEM, ResetClass := E_ResetClass.AUTO_RESET);
END_IF
IF auditSlot > 0 THEN AlarmLog.Gone(Slot := auditSlot); END_IF
END_METHOD

// §7.6.1 — concrete Units override to map a target path to a child module and call
// its ManualCommand. Base returns FALSE (no commandable children).
METHOD PROTECTED _M_RouteManual : BOOL
VAR_INPUT
    TargetPath : STRING(255);
    Value : DINT;
END_VAR
_M_RouteManual := FALSE;
END_METHOD

// §3.4.1/§3.14.4 — default per-mode switch policy. Station config (§3.8a) may
// overwrite ModePolicy[] after this. By FRAMEWORK DEFAULT a mode change while a
// sequence runs performs an IMMEDIATE software abort (E-stop-like, not a safety
// function, §3.14.4) — so Style defaults to IMMEDIATE. GRACEFUL completion is an
// opt-in: a Unit overrides OnModeExit to stop-after-cycle, or station config sets
// Style := GRACEFUL for a mode. Shield only governs acceptance while running.
METHOD PROTECTED _M_InitModePolicy
VAR
    i : INT;
END_VAR
FOR i := 0 TO PL_Fraktal.MODE_COUNT-1 DO
    ModePolicy[i].Shield := E_ModeSwitchShield.CONFIRM;
    ModePolicy[i].Style  := E_ModeSwitchStyle.IMMEDIATE;
END_FOR
// Setup modes a running machine may not leave without an explicit Stop first.
ModePolicy[TO_INT(E_Mode.CHANGEOVER)].Shield := E_ModeSwitchShield.BLOCKED_WHILE_RUNNING;
ModePolicy[TO_INT(E_Mode.CALIBRATION)].Shield:= E_ModeSwitchShield.BLOCKED_WHILE_RUNNING;
// HOME and MANUAL are freely interruptible; both inherit the IMMEDIATE default.
ModePolicy[TO_INT(E_Mode.HOME)].Shield       := E_ModeSwitchShield.INTERRUPTIBLE;
ModePolicy[TO_INT(E_Mode.MANUAL)].Shield     := E_ModeSwitchShield.INTERRUPTIBLE;
END_METHOD

// §3.4.2 — HMI selects the run style for the active mode. Modes that don't opt in
// (see _M_SupportsRunStyle) reject non-CONTINUOUS. Access: MODE_CHANGE-gated (§7.7).
METHOD SetRunStyle : BOOL
VAR_INPUT
    Style : E_RunStyle;
END_VAR
IF NOT Access.PermitsLogged(Gate := E_GatedAction.MODE_CHANGE) THEN
    SetRunStyle := FALSE;
    RETURN;
END_IF
IF (Style <> E_RunStyle.CONTINUOUS) AND NOT _M_SupportsRunStyle(Style := Style) THEN
    SetRunStyle := FALSE;               // mode didn't opt into stepping (graceful reject)
    RETURN;
END_IF
RunStyle := Style;
SetRunStyle := TRUE;
END_METHOD

// §3.4.2 — a concrete Unit overrides to opt a mode into SINGLE_STEP/HOLD_TO_RUN.
// Base: only CONTINUOUS.
METHOD PROTECTED _M_SupportsRunStyle : BOOL
VAR_INPUT
    Style : E_RunStyle;
END_VAR
_M_SupportsRunStyle := (Style = E_RunStyle.CONTINUOUS);
END_METHOD

// §3.4.2 — HMI single-step: request advance of one step (edge-consumed by _M_StepGate).
METHOD StepRequest : BOOL
IF NOT Access.PermitsLogged(Gate := E_GatedAction.START_STOP)
OR (RunStyle <> E_RunStyle.SINGLE_STEP) OR (_exec <> E_ExecState.BUSY) THEN
    StepRequest := FALSE;
    RETURN;
END_IF
_stepReq := TRUE;
StepRequest := TRUE;
END_METHOD

// §3.4.2 — HMI HOLD_TO_RUN input. NON-SAFETY (§9): never a dead-man; interlocks
// still apply at every step. TRUE only while the operator holds the button.
METHOD SetHoldRun : BOOL
VAR_INPUT
    Held : BOOL;
END_VAR
IF Held AND (NOT Access.PermitsLogged(Gate := E_GatedAction.START_STOP)
OR (RunStyle <> E_RunStyle.HOLD_TO_RUN) OR (_exec <> E_ExecState.BUSY)) THEN
    SetHoldRun := FALSE;
    RETURN;
END_IF
_holdRun := Held;                     // FALSE is always accepted so a hold cannot stick
SetHoldRun := TRUE;
END_METHOD

// §3.4.2 — the sequence author calls this at each step boundary; returns TRUE when
// the sequence may advance. Steppable (default TRUE) is the PER-STEP stop-point flag:
// a step with Steppable := FALSE runs straight through even in SINGLE_STEP/HOLD_TO_RUN
// (group several motions into one operator step, or a step unsafe to pause mid-way).
// CONTINUOUS: always TRUE. SINGLE_STEP: TRUE once per StepRequest edge (only if
// Steppable). HOLD_TO_RUN: TRUE while held (only if Steppable). Interlocks are
// enforced by the modules regardless (this only paces the sequence).
METHOD PROTECTED _M_StepGate : BOOL
VAR_INPUT
    Steppable : BOOL;
END_VAR
IF NOT Steppable THEN
    _M_StepGate := TRUE;               // not a stop point: advance regardless of run style
    RETURN;
END_IF
CASE RunStyle OF
    E_RunStyle.SINGLE_STEP:
        _stepArm(CLK := _stepReq);
        _stepReq := FALSE;
        _M_StepGate := _stepArm.Q;      // one advance per request edge
    E_RunStyle.HOLD_TO_RUN:
        _M_StepGate := _holdRun;        // advance only while held (NON-SAFETY)
ELSE
    _M_StepGate := TRUE;                // CONTINUOUS
END_CASE
END_METHOD

// §3.4 — TRUE while a stop is requested but the sequence is still finishing
// (running -> stopping). HMI blinks the stop button on this.
PROPERTY StopPending : BOOL
GET
StopPending := _stopReq AND (_exec = E_ExecState.BUSY);
END_GET
END_PROPERTY

// Core §7.8 — pure query: the FULL rollup of why Start would be refused right now.
// This is the authoritative machine predicate consumed by Start (no drift).
// Released = TRUE means Start proceeds. Lists mode + access + blocking-alarm,
// control-domain, and concrete mode-entry release reasons. The caller owns the
// bounded report storage; returning this large record by value can overflow a
// TwinCAT task stack when Start consumes the result.
METHOD ReleaseReportStart : BOOL
VAR_IN_OUT
    Report : ST_ReleaseReport;
END_VAR
Report.Count := 0;
Report.Released := FALSE;
// access (§7.7)
IF NOT Access.Permits(Gate := E_GatedAction.START_STOP) THEN
    _M_AddReason(Report := Report, Text := 'std.release.insufficientStartStop', Reason := E_Reason.NONE, Kind := E_ReleaseKind.ACCESS);
END_IF
// mode / run state (§3.4)
IF _modePend THEN
    _M_AddReason(Report := Report, Text := 'std.release.modeChangePending', Reason := E_Reason.NONE, Kind := E_ReleaseKind.MODE);
END_IF
IF _mode = E_Mode.MANUAL THEN
    _M_AddReason(Report := Report, Text := 'std.release.manualHasNoAutoSequence', Reason := E_Reason.NONE, Kind := E_ReleaseKind.MODE);
END_IF
IF _exec <> E_ExecState.READY THEN
    _M_AddReason(Report := Report, Text := 'std.release.unitNotReady', Reason := E_Reason.NONE, Kind := E_ReleaseKind.MODE);
END_IF
// blocking alarm (§8.3)
IF AlarmLog.Blocking THEN
    _M_AddReason(Report := Report, Text := 'std.release.manualReset', Reason := E_Reason.NONE, Kind := E_ReleaseKind.ALARM);
END_IF
IF ControlDomain.Present AND NOT ControlDomain.ReadyForStart THEN
    _M_AddReason(Report := Report, Text := 'std.release.controlDomainNotReady', Reason := E_Reason.NONE, Kind := E_ReleaseKind.INTERLOCK);
END_IF
// active mode's immediate entry/frontier conditions (concrete override)
_M_AppendInterlocks(Report := Report);
Report.Released := (Report.Count = 0);
ReleaseReportStart := Report.Released;
END_METHOD

// Core §7.8 — full rollup of why a manual command to Target would be refused (§7.6.1).
METHOD ReleaseReportManual : BOOL
VAR_INPUT
    TargetPath : STRING(255);
    Value : DINT;
END_VAR
VAR_IN_OUT
    Report : ST_ReleaseReport;
END_VAR
Report.Count := 0;
Report.Released := FALSE;
IF _mode <> E_Mode.MANUAL THEN
    _M_AddReason(Report := Report, Text := 'std.release.manualModeRequired', Reason := E_Reason.NONE, Kind := E_ReleaseKind.MODE);
END_IF
IF NOT Access.Permits(Gate := E_GatedAction.MANUAL) THEN
    _M_AddReason(Report := Report, Text := 'std.release.insufficientManual', Reason := E_Reason.NONE, Kind := E_ReleaseKind.ACCESS);
END_IF
_M_AppendManualInterlocks(TargetPath := TargetPath, Value := Value, Report := Report);  // §7.6, target+command-aware
Report.Released := (Report.Count = 0);
ReleaseReportManual := Report.Released;
END_METHOD

// Core §7.8 — concrete Units override to append the active mode's immediate
// entry/frontier records via PermIntlk.AppendFailed(SourcePath, Report). Future step waits
// stay in CurrentStep/Pending and are not blanket Start conditions. Base: nothing.
METHOD PROTECTED _M_AppendInterlocks
VAR_IN_OUT
    Report : ST_ReleaseReport;
END_VAR
;
END_METHOD

// Core §7.8 helper — append one non-interlock reason (bounds-checked).
METHOD PROTECTED _M_AddReason
VAR_IN_OUT
    Report : ST_ReleaseReport;
END_VAR
VAR_INPUT
    Text : STRING(255);
    Reason : E_Reason;
    Kind : E_ReleaseKind;
END_VAR
IF Report.Count >= PL_Fraktal.MAX_RELEASE_REASONS THEN
    RETURN;
END_IF
Report.Count := Report.Count + 1;
Report.Reasons[Report.Count].Description := Text;
Report.Reasons[Report.Count].ReasonCode  := Reason;
Report.Reasons[Report.Count].SourcePath  := _name;
Report.Reasons[Report.Count].Kind        := Kind;
Report.Reasons[Report.Count].Bypassable  := FALSE;
END_METHOD

// Core §7.8 — full rollup for the simpler gated Unit actions (Stop, ALARM_RESET,
// CHANGEOVER, MODE_CHANGE, step). Same predicate the gates use. Start has its own
// richer ReleaseReportStart (interlocks); manual has ReleaseReportManual (target).
METHOD ReleaseReportAction : BOOL
VAR_INPUT
    Gate : E_GatedAction;
END_VAR
VAR_IN_OUT
    Report : ST_ReleaseReport;
END_VAR
Report.Count := 0;
Report.Released := FALSE;
// access is the common gate
IF NOT Access.Permits(Gate := Gate) THEN
    _M_AddReason(Report := Report, Text := 'std.release.insufficientAction', Reason := E_Reason.NONE, Kind := E_ReleaseKind.ACCESS);
END_IF
// per-action state preconditions
CASE Gate OF
    E_GatedAction.CHANGEOVER:
        IF _exec = E_ExecState.BUSY THEN
            _M_AddReason(Report := Report, Text := 'std.release.changeoverRunning', Reason := E_Reason.NONE, Kind := E_ReleaseKind.MODE);
        END_IF
    E_GatedAction.ALARM_RESET:
        IF NOT AlarmLog.Blocking THEN
            _M_AddReason(Report := Report, Text := 'std.release.noBlockingAlarm', Reason := E_Reason.NONE, Kind := E_ReleaseKind.OTHER);
        END_IF
    E_GatedAction.MODE_CHANGE:
        IF _modePend THEN
            _M_AddReason(Report := Report, Text := 'std.release.modeChangeAlreadyPending', Reason := E_Reason.NONE, Kind := E_ReleaseKind.MODE);
        END_IF
ELSE
    ;                                          // actions with no extra state predicate
END_CASE
Report.Released := (Report.Count = 0);
ReleaseReportAction := Report.Released;
END_METHOD

// §8.5.1 — attribute elapsed time to run/down/idle, recompute factors, sample ring.
METHOD PROTECTED _M_OeeUpdate
VAR
    currentTime : TIME;
    deltaMs     : UDINT;
END_VAR
currentTime := TIME();                 // monotonic duration clock
IF _oeeLast = T#0S THEN
    _oeeLast := currentTime;
    RETURN;
END_IF
deltaMs := TIME_TO_UDINT(currentTime) - TIME_TO_UDINT(_oeeLast); // wrap-safe on UDINT subtraction
_oeeLast := currentTime;
IF _exec = E_ExecState.BUSY THEN
    Oee.RunMs := Oee.RunMs + deltaMs;
ELSIF (_exec = E_ExecState.ERROR) OR AlarmLog.Blocking THEN
    Oee.DownMs := Oee.DownMs + deltaMs;
ELSE
    Oee.IdleMs := Oee.IdleMs + deltaMs;
END_IF
_M_OeeCompute();
_oeeSampMs := _oeeSampMs + deltaMs;
IF _oeeSampMs >= PL_Fraktal.OEE_SAMPLE_MS THEN
    _oeeSampMs := 0;
    OeeTrendHead := (OeeTrendHead MOD PL_Fraktal.MAX_OEE_SAMPLES) + 1;
    OeeTrend[OeeTrendHead].Availability := Oee.Availability;
    OeeTrend[OeeTrendHead].Performance  := Oee.Performance;
    OeeTrend[OeeTrendHead].Quality      := Oee.Quality;
    OeeTrend[OeeTrendHead].Oee          := Oee.Oee;
    OeeTrend[OeeTrendHead].OeeValid     := Oee.OeeValid;
END_IF
END_METHOD

// §8.5.1 — pure recompute of A/P/Q/OEE from the accumulators (testable in isolation).
// Invalid factors are OMITTED from the product, never assumed 100% (O7).
METHOD PROTECTED _M_OeeCompute
VAR
    total : UDINT;
    denomA: UDINT;
END_VAR
denomA := Oee.RunMs + Oee.DownMs;
Oee.AvailValid := denomA > 0;
IF Oee.AvailValid THEN
    Oee.Availability := UDINT_TO_REAL(Oee.RunMs) / UDINT_TO_REAL(denomA);
ELSE
    Oee.Availability := 0.0;
END_IF
Oee.PerfValid := (Oee.IdealCycleMs > 0) AND (Oee.RunMs > 0);
IF Oee.PerfValid THEN
    Oee.Performance := UDINT_TO_REAL(Oee.IdealCycleMs) * UDINT_TO_REAL(GoodCount + NokCount)
                       / UDINT_TO_REAL(Oee.RunMs);
    IF Oee.Performance > 1.0 THEN
        Oee.Performance := 1.0;          // faster than ideal caps at 100% (standard practice)
    END_IF
ELSE
    Oee.Performance := 0.0;
END_IF
total := GoodCount + NokCount;
Oee.QualValid := total > 0;
IF Oee.QualValid THEN
    Oee.Quality := UDINT_TO_REAL(GoodCount) / UDINT_TO_REAL(total);
ELSE
    Oee.Quality := 0.0;
END_IF
// product of VALID factors only; OEE valid iff at least one factor is valid
Oee.Oee := 1.0;
Oee.OeeValid := FALSE;
IF Oee.AvailValid THEN Oee.Oee := Oee.Oee * Oee.Availability; Oee.OeeValid := TRUE; END_IF
IF Oee.PerfValid  THEN Oee.Oee := Oee.Oee * Oee.Performance;  Oee.OeeValid := TRUE; END_IF
IF Oee.QualValid  THEN Oee.Oee := Oee.Oee * Oee.Quality;      Oee.OeeValid := TRUE; END_IF
IF NOT Oee.OeeValid THEN
    Oee.Oee := 0.0;
END_IF
END_METHOD

// §8.5.1 — configure the ideal cycle time (per model, §3.8). 0 disables Performance.
METHOD SetIdealCycle : BOOL
VAR_INPUT
    Ms : UDINT;
END_VAR
Oee.IdealCycleMs := Ms;
SetIdealCycle := TRUE;
END_METHOD

// §8.5.1 — clear accumulators + ring (shift start). Gated: §7.7 DATA_WRITE; audited §8.3.
METHOD ResetOee : BOOL
VAR
    i : INT;
    auditSlot : INT;
END_VAR
IF NOT Access.PermitsLogged(Gate := E_GatedAction.DATA_WRITE) THEN
    ResetOee := FALSE;
    RETURN;
END_IF
Oee.RunMs := 0; Oee.DownMs := 0; Oee.IdleMs := 0;
FOR i := 1 TO PL_Fraktal.MAX_OEE_SAMPLES DO
    OeeTrend[i].Oee := 0.0; OeeTrend[i].OeeValid := FALSE;
    OeeTrend[i].Availability := 0.0; OeeTrend[i].Performance := 0.0; OeeTrend[i].Quality := 0.0;
END_FOR
OeeTrendHead := 0;
_oeeSampMs := 0;
_M_OeeCompute();
auditSlot := AlarmLog.Raise(Reason := E_Reason.NONE,
    Text := 'std.audit.oeeReset', Source := _name,
    Severity := E_Severity.LOW, Category := E_Category.SYSTEM, ResetClass := E_ResetClass.AUTO_RESET);
IF auditSlot > 0 THEN AlarmLog.Gone(Slot := auditSlot); END_IF
ResetOee := TRUE;
END_METHOD

// §8.10 — gated HMI entry: shelve an active alarm's ANNUNCIATION (control untouched).
// §7.7 ALARM_SHELVE + audit; refuses SAFETY / unrationalized reasons (AlarmLog rules).
METHOD ShelveAlarm : BOOL
VAR_INPUT
    Slot      : INT;
    DurationS : UDINT;
END_VAR
IF NOT Access.PermitsLogged(Gate := E_GatedAction.ALARM_SHELVE) THEN
    ShelveAlarm := FALSE;
    RETURN;
END_IF
ShelveAlarm := AlarmLog.Shelve(Slot := Slot, DurationS := DurationS);
END_METHOD

// §8.10 — gated HMI entry: restore annunciation.
METHOD UnshelveAlarm : BOOL
VAR_INPUT
    Slot : INT;
END_VAR
IF NOT Access.PermitsLogged(Gate := E_GatedAction.ALARM_SHELVE) THEN
    UnshelveAlarm := FALSE;
    RETURN;
END_IF
UnshelveAlarm := AlarmLog.Unshelve(Slot := Slot);
END_METHOD

// Core §7.8 — target-aware hook for the MANUAL release rollup: a concrete Unit
// overrides to append the §7.6 Release<Function> conditions of the SPECIFIC target
// module. Base delegates to the Unit-level hook (non-breaking default).
METHOD PROTECTED _M_AppendManualInterlocks
VAR_INPUT
    TargetPath : STRING(255);
    Value : DINT;
END_VAR
VAR_IN_OUT
    Report : ST_ReleaseReport;
END_VAR
_M_AppendInterlocks(Report := Report);
END_METHOD

// §3.10/§14 — consume one committed OPC UA request exactly once.
METHOD PROTECTED _M_HandleHmiRequest
VAR
    modelId  : ST_ModelId;
    modeReq  : E_Mode;
    styleReq : E_RunStyle;
    gateReq  : E_GatedAction;
END_VAR
IF HmiRequest.Sequence = _hmiLastSequence THEN
    RETURN;
ELSE
    _hmiLastSequence := HmiRequest.Sequence;
END_IF

HmiResponse.Accepted := FALSE;
HmiResponse.Diagnostic := '';
HmiResponse.Report.Count := 0;
HmiResponse.Report.Released := FALSE;

CASE HmiRequest.Kind OF
    E_HmiRequestKind.LOGIN:
        HmiResponse.Accepted := Access.RequestLogin(User := HmiRequest.User, Secret := HmiRequest.Secret);
    E_HmiRequestKind.LOGOUT:
        HmiResponse.Accepted := Access.RequestLogout();
    E_HmiRequestKind.SET_MODE:
        IF (HmiRequest.IntValue >= 0) AND (HmiRequest.IntValue < PL_Fraktal.MODE_COUNT) THEN
            modeReq := HmiRequest.IntValue;
            HmiResponse.Accepted := SetMode(Mode := modeReq);
        ELSE
            HmiResponse.Diagnostic := 'std.error.unsupportedModeRequest';
        END_IF
    E_HmiRequestKind.SET_MODEL:
        modelId.ModelCode := HmiRequest.TextValue;
        HmiResponse.Accepted := SetModel(Id := modelId);
    E_HmiRequestKind.START:
        HmiResponse.Accepted := Start();
    E_HmiRequestKind.STOP:
        HmiResponse.Accepted := Stop();
    E_HmiRequestKind.CONTROL_ON:
        ReqControlOn := TRUE;
        ReqControlOff := FALSE;
        HmiResponse.Accepted := TRUE;
    E_HmiRequestKind.CONTROL_OFF:
        ReqControlOff := TRUE;
        ReqControlOn := FALSE;
        HmiResponse.Accepted := TRUE;
    E_HmiRequestKind.OPERATOR_RESET:
        HmiResponse.Accepted := OperatorReset();
    E_HmiRequestKind.DECISION_ANSWER:
        DecisionAnswer := TO_INT(HmiRequest.IntValue);
        HmiResponse.Accepted := TRUE;
    E_HmiRequestKind.MANUAL_COMMAND:
        HmiResponse.Accepted := ManualCommandTo(TargetPath := HmiRequest.TargetPath, Value := HmiRequest.IntValue);
    E_HmiRequestKind.SET_RUN_STYLE:
        IF (HmiRequest.IntValue >= 0) AND (HmiRequest.IntValue <= 2) THEN
            styleReq := HmiRequest.IntValue;
            HmiResponse.Accepted := SetRunStyle(Style := styleReq);
        ELSE
            HmiResponse.Diagnostic := 'std.error.unsupportedRunStyleRequest';
        END_IF
    E_HmiRequestKind.STEP_REQUEST:
        HmiResponse.Accepted := StepRequest();
    E_HmiRequestKind.SET_HOLD_RUN:
        HmiResponse.Accepted := SetHoldRun(Held := HmiRequest.BoolValue);
    E_HmiRequestKind.RELEASE_START:
        ReleaseReportStart(Report := HmiResponse.Report);
        HmiResponse.Accepted := TRUE;
    E_HmiRequestKind.RELEASE_MANUAL:
        ReleaseReportManual(TargetPath := HmiRequest.TargetPath, Value := HmiRequest.IntValue,
            Report := HmiResponse.Report);
        HmiResponse.Accepted := TRUE;
    E_HmiRequestKind.RELEASE_ACTION:
        IF (HmiRequest.IntValue >= 0) AND (HmiRequest.IntValue <= 10) THEN
            gateReq := HmiRequest.IntValue;
            ReleaseReportAction(Gate := gateReq, Report := HmiResponse.Report);
            HmiResponse.Accepted := TRUE;
        ELSE
            HmiResponse.Diagnostic := 'std.error.unsupportedGatedActionRequest';
        END_IF
    E_HmiRequestKind.RESET_OEE:
        HmiResponse.Accepted := ResetOee();
    E_HmiRequestKind.WRITE_CONFIG:
        HmiResponse.Accepted := _M_RouteConfigWrite(TargetPath := HmiRequest.TargetPath,
            FieldName := HmiRequest.NameValue, TextValue := HmiRequest.TextValue);
    E_HmiRequestKind.SHELVE_ALARM:
        HmiResponse.Diagnostic := 'std.error.identityAlarmRequestNotSupported';
    E_HmiRequestKind.UNSHELVE_ALARM:
        HmiResponse.Diagnostic := 'std.error.identityAlarmRequestNotSupported';
    E_HmiRequestKind.FORCE_CHANNEL:
        HmiResponse.Accepted := _M_RouteForceChannel(ChannelPath := HmiRequest.TargetPath,
            Force := HmiRequest.BoolValue, BoolText := HmiRequest.TextValue,
            AnalogText := HmiRequest.NameValue);
    E_HmiRequestKind.NONE:
        HmiResponse.Diagnostic := 'std.error.emptyHmiRequest';
ELSE
    HmiResponse.Diagnostic := 'std.error.unsupportedHmiRequest';
END_CASE

IF NOT HmiResponse.Accepted AND (HmiResponse.Diagnostic = '') THEN
    HmiResponse.Diagnostic := 'std.error.hmiRequestRejected';
ELSE
    HmiResponse.Diagnostic := HmiResponse.Diagnostic;
END_IF
HmiRequest.Secret := '';
HmiResponse.AckSequence := _hmiLastSequence;
END_METHOD

// Project/type override for published editable fields. Base fails closed.
METHOD PROTECTED _M_RouteConfigWrite : BOOL
VAR_INPUT
    TargetPath : STRING(255);
    FieldName  : STRING(160);
    TextValue  : STRING(255);
END_VAR
_M_RouteConfigWrite := FALSE;
END_METHOD

// Application override routes only approved outputs through its force gate.
METHOD PROTECTED _M_RouteForceChannel : BOOL
VAR_INPUT
    ChannelPath : STRING(255);
    Force       : BOOL;
    BoolText    : STRING(255);
    AnalogText  : STRING(160);
END_VAR
_M_RouteForceChannel := FALSE;
END_METHOD

END_FUNCTION_BLOCK

// ---- Connectivity/FB_DeviceConnectorBase.TcPOU
// Core §3.15 written once: session + heartbeat + LinkTimeout loss confirm +
// bounded exponential backoff reconnect + NO self-resume of dependents (that is
// the fronting CM's contract). A transport implements only _M_Open/_M_Close/
// _M_HbStart/_M_HbPoll. Row T7 of §5.7 is proven here once.
{attribute 'OPC.UA.DA' := '1'}
FUNCTION_BLOCK ABSTRACT FB_DeviceConnectorBase IMPLEMENTS I_DeviceConnector
VAR_INPUT
    HbPeriod    : TIME := T#1S;
    LinkTimeout : TIME := T#3S;
    BackoffMin  : TIME := T#500MS;
    BackoffMax  : TIME := T#10S;
    Reaction    : E_LinkReaction := E_LinkReaction.HOLD;   // consumed by the fronting CM
END_VAR
VAR
    _name      : STRING(80);
    _sessionUp : BOOL;
    _linked    : BOOL;
    _hbBusy    : BOOL;
    _lastSeen  : DT;
    _diag      : ST_Diagnostic;
    _tHb, _tLoss, _tBk : TON;
    _backoffMs : DINT;
END_VAR

Cyclic();

METHOD Connect : BOOL
Connect := _M_TryOpen();
END_METHOD

METHOD Cyclic : BOOL
IF NOT _sessionUp THEN
    // bounded exponential backoff (§3.15) — never a tight reconnect loop
    _tBk(IN := TRUE, PT := DINT_TO_TIME(_backoffMs));
    IF _tBk.Q THEN
        _tBk(IN := FALSE);
        IF NOT _M_TryOpen() THEN
            _backoffMs := MIN(_backoffMs * 2, TIME_TO_DINT(BackoffMax));
        END_IF
    END_IF
    Cyclic := TRUE;
    RETURN;
END_IF
// heartbeat: issue when due, poll while busy
IF NOT _hbBusy THEN
    _tHb(IN := TRUE, PT := HbPeriod);
    IF _tHb.Q THEN
        _tHb(IN := FALSE);
        _hbBusy := _M_HbStart();
    END_IF
ELSE
    CASE _M_HbPoll() OF
        E_HbResult.OK:
            _hbBusy := FALSE;
            _linked := TRUE;
            _lastSeen := F_Now();                 // §2.7
            _diag.ReasonCode := E_Reason.NONE;
            _diag.Description := '';
            _tLoss(IN := FALSE);                  // healthy beat resets loss confirm
        E_HbResult.FAIL:
            _hbBusy := FALSE;
            _M_Lost(E_Reason.DEVICE_PROTOCOL_ERROR, 'std.error.heartbeatBadReply');
            Cyclic := TRUE;
            RETURN;
        E_HbResult.PENDING:
            ;                                      // request still in flight
    ELSE
        _hbBusy := FALSE;
        _M_Lost(E_Reason.DEVICE_PROTOCOL_ERROR, 'std.error.heartbeatResultInvalid');
        Cyclic := TRUE;
        RETURN;
    END_CASE
END_IF
// confirm loss only after LinkTimeout without a healthy beat (§3.15.2)
_tLoss(IN := TRUE, PT := LinkTimeout);
IF _tLoss.Q THEN
    _M_Lost(E_Reason.LINK_TIMEOUT, 'std.error.heartbeatLapsed');
END_IF
Cyclic := TRUE;
END_METHOD

METHOD Disconnect : BOOL
_M_Close();
_sessionUp := FALSE;
_linked := FALSE;
Disconnect := TRUE;
END_METHOD

METHOD GetFaultSummary : ST_Diagnostic
GetFaultSummary := _diag;
END_METHOD

METHOD PrepareRecipe : BOOL
VAR_INPUT
    Model : ST_ModelId;
END_VAR
PrepareRecipe := TRUE;
END_METHOD

METHOD CommitRecipe
END_METHOD

METHOD AbortRecipe
END_METHOD

METHOD Setup : BOOL
VAR_INPUT
    Name : STRING(80);
END_VAR
_name := Name;
_backoffMs := TIME_TO_DINT(BackoffMin);
Setup := TRUE;
END_METHOD

METHOD PROTECTED ABSTRACT _M_Close : BOOL
END_METHOD

// PENDING while in flight; OK resets loss confirm; FAIL = protocol error
METHOD PROTECTED ABSTRACT _M_HbPoll : E_HbResult
END_METHOD

METHOD PROTECTED ABSTRACT _M_HbStart : BOOL
END_METHOD

// stamp the link first-out, drop the session; reconnection is backoff-bounded,
// resumption of dependent commands is NEVER automatic (§3.15/§9.3)
METHOD PROTECTED _M_Lost
VAR_INPUT
    Reason : E_Reason;
    Text   : STRING(255);
END_VAR
IF _diag.ReasonCode <> Reason THEN
    _diag.Since := F_Now();
END_IF
_diag.ReasonCode  := Reason;
_diag.Description := Text;
_diag.SourcePath  := _name;
_diag.Severity    := E_Severity.MED;
_diag.Category    := E_Category.SYSTEM;
_linked := FALSE;
_hbBusy := FALSE;
_M_Close();
_sessionUp := FALSE;
END_METHOD

METHOD PROTECTED ABSTRACT _M_Open : BOOL
END_METHOD

METHOD PROTECTED _M_TryOpen : BOOL
IF _M_Open() THEN
    _sessionUp := TRUE;
    _backoffMs := TIME_TO_DINT(BackoffMin);
    _M_TryOpen := TRUE;
ELSE
    _M_TryOpen := FALSE;
END_IF
END_METHOD

PROPERTY FaultActive : BOOL
GET
FaultActive := (NOT _linked) AND (_diag.ReasonCode <> E_Reason.NONE);
END_GET
END_PROPERTY

PROPERTY LastSeen : DT
GET
LastSeen := _lastSeen;
END_GET
END_PROPERTY

PROPERTY Linked : BOOL
GET
Linked := _linked;
END_GET
END_PROPERTY

PROPERTY LinkReason : ST_Diagnostic
GET
LinkReason := _diag;
END_GET
END_PROPERTY

PROPERTY ModuleType : E_ModuleType
GET
ModuleType := E_ModuleType.CONTROL_MODULE;
END_GET
END_PROPERTY

PROPERTY Name : STRING(80)
GET
Name := _name;
END_GET
END_PROPERTY

PROPERTY State : E_ExecState
GET
State := SEL(FaultActive, E_ExecState.READY, E_ExecState.ERROR);
END_GET
END_PROPERTY

END_FUNCTION_BLOCK

// ---- Connectivity/FB_EcFieldbusScanner.TcPOU
// [TC3] SKELETON — default EtherCAT implementation of I_FieldbusScanner (TC3 §10.6).
// This is a CONTRACT SKELETON: the structure and the Tc2_EtherCAT building blocks
// are named; bodies are TODO for the integrator, who must verify every index group,
// port, and FB signature against the pinned Tc2_EtherCAT version (Beckhoff InfoSys).
// See fraktal-tc3/FIELDBUS_ADS_ADAPTER.md for the full contract and the AL-state map.
{attribute 'OPC.UA.DA' := '1'}
FUNCTION_BLOCK FB_EcFieldbusScanner IMPLEMENTS I_FieldbusScanner
VAR
    MasterNetId : STRING(23);        // EtherCAT master AmsNetId (from the master's ADS tab)
END_VAR
VAR
    // Tc2_EtherCAT building blocks (uncomment when the library is referenced):
    // _getCount   : FB_EcGetSlaveCount;         // slave count
    // _getStates  : FB_EcGetAllSlaveStates;     // bulk AL states (INIT/PREOP/SAFEOP/OP)
    // _getIdent   : FB_EcGetSlaveIdentity;      // vendor/product per slave
    // _coeRead    : FB_CoeSdoReadEx;            // CoE object dictionary (names, scaling)
    _slaveCount : INT;
END_VAR

// no cyclic body — driven via the interface methods by the owning application

METHOD Scan : INT
VAR_IN_OUT
    Data : ST_FieldbusTopology;
END_VAR
// TODO(integrator):
//  1) _getCount(sNetId := MasterNetId, ...) -> _slaveCount  (0 => master down => RETURN 0)
//  2) _getStates(...) -> per-slave AL state word; map with _M_MapState() into Nodes[i].State
//  3) _getIdent(...) per slave -> Nodes[i].TypeId / Address; set ParentIdx from topology order
//  4) per slave, discover channels: CoE object dictionary (_coeRead of 0x6000/0x7000 ranges)
//     OR the configured PDO mapping -> fill Nodes[i].Channels[].Name/Dir/Kind/Unit
//  Verify index groups/ports against Tc2_EtherCAT InfoSys before trusting any value.
Scan := 0;   // skeleton: returns 'master down' until implemented
END_METHOD

METHOD RefreshValues : BOOL
VAR_IN_OUT
    Data : ST_FieldbusTopology;
END_VAR
// TODO(integrator): copy live values from the PLC PROCESS IMAGE (the variables the
// terminals are linked to) into Nodes[i].Channels[j].BoolValue/AnalogValue/Quality.
// PREFERRED: the application links each channel to the HAL struct it already owns
// (§3.6) and sets a pointer/reference here — no raw process-image address math.
// Analog scaling (raw INT -> REAL + Unit) comes from the ESI/TMC or the CM's ParCfg.
RefreshValues := FALSE;
END_METHOD

METHOD ForceChannel : BOOL
VAR_INPUT
    ChannelPath : STRING(255);
    Force       : BOOL;
    BoolValue   : BOOL;
    AnalogRaw   : DINT;
END_VAR
// OUTPUT-ONLY force (Core §10.5.1 rule): write the MAPPED OUTPUT VARIABLE for the
// channel. Reject inputs and unknown channels. This is NOT a raw process-image
// force and cannot touch inputs or safety I/O. Caller has ALREADY checked
// §7.6/§7.7 and will log the §8.3 event; do NOT re-gate here.
// TODO(integrator):
//  1) resolve ChannelPath -> the owning module's HAL output field (via the same
//     reference table RefreshValues uses); if not found OR it is an input -> FALSE.
//  2) Force=TRUE  -> latch BoolValue/AnalogRaw onto that output each scan while held;
//     Force=FALSE -> release (module resumes driving it).
// Because the write goes through the application, a RUNNING module reasserts its
// own output — a force is only effective when the module is stopped/in MANUAL,
// which is the intended safety behaviour (the force cannot override active logic).
ForceChannel := FALSE;   // skeleton: rejects until implemented
END_METHOD

// EtherCAT AL-state word -> neutral E_NodeState (Core §10.5.1). The AL-state low
// nibble is the state; bit 0x10 is the error/fault flag. VERIFY constants (InfoSys).
METHOD PROTECTED _M_MapState : E_NodeState
VAR_INPUT
    AlState : WORD;
END_VAR
VAR
    stateNibble : WORD;
END_VAR
IF (AlState AND 16#0010) <> 0 THEN
    _M_MapState := E_NodeState.FAULT;               // AL error bit set
    RETURN;
END_IF
stateNibble := AlState AND 16#000F;
CASE stateNibble OF
    16#01: _M_MapState := E_NodeState.INIT;
    16#02: _M_MapState := E_NodeState.PREOP;
    16#04: _M_MapState := E_NodeState.SAFEOP;
    16#08: _M_MapState := E_NodeState.OPERATIONAL;
ELSE
    _M_MapState := E_NodeState.OFFLINE;             // incl. BOOTSTRAP(0x03)/no-response
END_CASE
END_METHOD

END_FUNCTION_BLOCK

// ---- Connectivity/FB_IoTopologyPublisher.TcPOU
// Core §10.5.1 infrastructure service. Owns the reusable bounded-table,
// validation, health and diagnostic-join algorithms; project code supplies only
// physical topology metadata and live values. This is not a module tier.
FUNCTION_BLOCK FB_IoTopologyPublisher
VAR
    _data : REFERENCE TO ST_FieldbusTopology;
    _attached : BOOL;
END_VAR

;

METHOD Setup : BOOL
VAR_INPUT
    DataRef : REFERENCE TO ST_FieldbusTopology;
    ResetData : BOOL;
END_VAR
VAR
    n, c : INT;
END_VAR
_data REF= DataRef;
_attached := __ISVALIDREF(_data);
IF _attached AND ResetData THEN
    _data.NodeCount := 0;
    _data.MappingValid := TRUE;
    _data.MappingDiagnostic := '';
    FOR n := 1 TO PL_Fraktal.MAX_BUS_NODES DO
        _data.Nodes[n].Name := '';
        _data.Nodes[n].DescriptionKey := '';
        _data.Nodes[n].TypeId := '';
        _data.Nodes[n].Address := '';
        _data.Nodes[n].ParentIdx := 0;
        _data.Nodes[n].ChannelCount := 0;
        FOR c := 1 TO PL_Fraktal.MAX_NODE_CHANNELS DO
            _data.Nodes[n].Channels[c].Name := '';
            _data.Nodes[n].Channels[c].Path := '';
        END_FOR
    END_FOR
ELSIF _attached THEN
    ;
ELSE
    _attached := FALSE;
END_IF
Setup := _attached;
END_METHOD

METHOD M_DefineNode : BOOL
VAR_INPUT
    Index : INT;
    Name : STRING(80);
    DescriptionKey : STRING(160);
    TypeId : STRING(80);
    Address : STRING(40);
    ParentIndex : INT;
END_VAR
M_DefineNode := FALSE;
IF NOT _attached THEN
    RETURN;
ELSE
    ;
END_IF
IF (Index < 1) OR (Index > PL_Fraktal.MAX_BUS_NODES)
OR (Name = '') OR (Address = '')
OR (ParentIndex < 0) OR (ParentIndex >= Index) THEN
    _M_Reject(Text := 'std.error.fieldbusNodeMappingInvalid');
    RETURN;
ELSE
    ;
END_IF
_data.Nodes[Index].Name := Name;
_data.Nodes[Index].DescriptionKey := DescriptionKey;
_data.Nodes[Index].TypeId := TypeId;
_data.Nodes[Index].Address := Address;
_data.Nodes[Index].ParentIdx := ParentIndex;
IF Index > _data.NodeCount THEN
    _data.NodeCount := Index;
ELSE
    ;
END_IF
M_DefineNode := TRUE;
END_METHOD

METHOD M_DefineDigitalChannel : BOOL
VAR_INPUT
    NodeIndex : INT;
    ChannelIndex : INT;
    Tag : STRING(80);
    DescriptionKey : STRING(160);
    Address : STRING(80);
    Path : STRING(255);
    ModulePath : STRING(255);
    Dir : E_ChannelDir;
END_VAR
M_DefineDigitalChannel := FALSE;
IF NOT _attached THEN
    RETURN;
ELSE
    ;
END_IF
IF (NodeIndex < 1) OR (NodeIndex > _data.NodeCount)
OR (ChannelIndex < 1) OR (ChannelIndex > PL_Fraktal.MAX_NODE_CHANNELS)
OR (Tag = '') OR (DescriptionKey = '') OR (Address = '')
OR (Path = '') OR (ModulePath = '') THEN
    _M_Reject(Text := 'std.error.fieldbusChannelMappingInvalid');
    RETURN;
ELSE
    ;
END_IF
_data.Nodes[NodeIndex].Channels[ChannelIndex].Name := Tag;
_data.Nodes[NodeIndex].Channels[ChannelIndex].DescriptionKey := DescriptionKey;
_data.Nodes[NodeIndex].Channels[ChannelIndex].Address := Address;
_data.Nodes[NodeIndex].Channels[ChannelIndex].Path := Path;
_data.Nodes[NodeIndex].Channels[ChannelIndex].ModulePath := ModulePath;
_data.Nodes[NodeIndex].Channels[ChannelIndex].Dir := Dir;
_data.Nodes[NodeIndex].Channels[ChannelIndex].Kind := E_ChannelKind.DIGITAL;
_data.Nodes[NodeIndex].Channels[ChannelIndex].Quality := TRUE;
IF ChannelIndex > _data.Nodes[NodeIndex].ChannelCount THEN
    _data.Nodes[NodeIndex].ChannelCount := ChannelIndex;
ELSE
    ;
END_IF
M_DefineDigitalChannel := TRUE;
END_METHOD

METHOD M_SetDigitalValue : BOOL
VAR_INPUT
    NodeIndex : INT;
    ChannelIndex : INT;
    Value : BOOL;
END_VAR
M_SetDigitalValue := FALSE;
IF _attached AND (NodeIndex >= 1) AND (NodeIndex <= _data.NodeCount)
AND (ChannelIndex >= 1) AND (ChannelIndex <= _data.Nodes[NodeIndex].ChannelCount) THEN
    _data.Nodes[NodeIndex].Channels[ChannelIndex].BoolValue := Value;
    M_SetDigitalValue := TRUE;
ELSE
    _M_Reject(Text := 'std.error.fieldbusValueMappingInvalid');
END_IF
END_METHOD

METHOD M_SetAllHealth
VAR_INPUT
    Healthy : BOOL;
END_VAR
VAR
    n, c : INT;
END_VAR
IF _attached THEN
    FOR n := 1 TO _data.NodeCount DO
        _data.Nodes[n].LinkOk := Healthy;
        IF Healthy THEN
            _data.Nodes[n].State := E_NodeState.OPERATIONAL;
        ELSE
            _data.Nodes[n].State := E_NodeState.FAULT;
        END_IF
        FOR c := 1 TO _data.Nodes[n].ChannelCount DO
            _data.Nodes[n].Channels[c].Quality := Healthy;
        END_FOR
    END_FOR
ELSE
    ;
END_IF
END_METHOD

METHOD M_BeginDiagnosticRefresh
VAR
    n, c : INT;
END_VAR
IF _attached THEN
    FOR n := 1 TO _data.NodeCount DO
        FOR c := 1 TO _data.Nodes[n].ChannelCount DO
            _data.Nodes[n].Channels[c].FaultActive := FALSE;
            _data.Nodes[n].Channels[c].Diagnostic := '';
        END_FOR
    END_FOR
ELSE
    ;
END_IF
END_METHOD

METHOD M_ApplyDiagnostic
VAR_INPUT
    Diagnostic : ST_Diagnostic;
END_VAR
IF Diagnostic.IoTag <> '' THEN
    M_ApplyDiagnosticToTag(Diagnostic := Diagnostic, Tag := Diagnostic.IoTag);
ELSE
    ;
END_IF
END_METHOD

METHOD M_ApplyDiagnosticToTag
VAR_INPUT
    Diagnostic : ST_Diagnostic;
    Tag : STRING(80);
END_VAR
VAR
    n, c : INT;
END_VAR
IF _attached AND (Tag <> '') THEN
    FOR n := 1 TO _data.NodeCount DO
        FOR c := 1 TO _data.Nodes[n].ChannelCount DO
            IF _data.Nodes[n].Channels[c].Name = Tag THEN
                _data.Nodes[n].Channels[c].FaultActive := TRUE;
                _data.Nodes[n].Channels[c].Diagnostic := Diagnostic.Description;
            ELSE
                ;
            END_IF
        END_FOR
    END_FOR
ELSE
    ;
END_IF
END_METHOD

METHOD M_Validate : BOOL
VAR
    n, c, n2, c2 : INT;
END_VAR
M_Validate := FALSE;
IF NOT _attached OR (_data.NodeCount < 1) THEN
    _M_Reject(Text := 'std.error.fieldbusTopologyEmpty');
    RETURN;
ELSE
    ;
END_IF
IF NOT _data.MappingValid THEN
    RETURN; // preserve the first registration/value mapping failure
ELSE
    ;
END_IF
FOR n := 1 TO _data.NodeCount DO
    IF (_data.Nodes[n].Name = '') OR (_data.Nodes[n].Address = '') THEN
        _M_Reject(Text := 'std.error.fieldbusNodeMappingInvalid');
        RETURN;
    ELSE
        ;
    END_IF
    FOR c := 1 TO _data.Nodes[n].ChannelCount DO
        IF (_data.Nodes[n].Channels[c].Name = '')
        OR (_data.Nodes[n].Channels[c].Address = '')
        OR (_data.Nodes[n].Channels[c].Path = '')
        OR (_data.Nodes[n].Channels[c].ModulePath = '') THEN
            _M_Reject(Text := 'std.error.fieldbusChannelMappingInvalid');
            RETURN;
        ELSE
            ;
        END_IF
        FOR n2 := n TO _data.NodeCount DO
            FOR c2 := 1 TO _data.Nodes[n2].ChannelCount DO
                IF ((n2 > n) OR (c2 > c))
                AND ((_data.Nodes[n].Channels[c].Name = _data.Nodes[n2].Channels[c2].Name)
                  OR (_data.Nodes[n].Channels[c].Path = _data.Nodes[n2].Channels[c2].Path)) THEN
                    _M_Reject(Text := 'std.error.fieldbusChannelIdentityDuplicate');
                    RETURN;
                ELSE
                    ;
                END_IF
            END_FOR
        END_FOR
    END_FOR
END_FOR
_data.MappingValid := TRUE;
_data.MappingDiagnostic := '';
M_Validate := TRUE;
END_METHOD

METHOD PRIVATE _M_Reject
VAR_INPUT
    Text : STRING(255);
END_VAR
IF _attached THEN
    _data.MappingValid := FALSE;
    _data.MappingDiagnostic := Text;
ELSE
    ;
END_IF
END_METHOD

END_FUNCTION_BLOCK

// ---- Connectivity/FB_LocalPartCarrier.TcPOU
// Core §3.16.2 — DEFAULT local carrier: BY_POSITION identity for stations without
// RFID/scanner/host. ReadContext assigns the next station-local serial from a
// configured prefix; WriteResult keeps a bounded ring of produced results so the
// HMI/MES adapter can collect them. RFID/DataMatrix/host carriers substitute
// behind I_PartCarrier later (the recipe-provider pattern, §3.8).
FUNCTION_BLOCK FB_LocalPartCarrier IMPLEMENTS I_PartCarrier
VAR_OUTPUT
    Produced     : ARRAY[1..PL_Fraktal.MAX_RECIPES] OF ST_PartResult; // last results ring
    ProducedHead : INT;                                               // newest entry (0 = none)
    ProducedUids : ARRAY[1..PL_Fraktal.MAX_RECIPES] OF STRING(64);
END_VAR
VAR
    _prefix : STRING(40);
    _serial : UDINT;
    _configured : BOOL;
END_VAR

// no cyclic body

// commissioning-time identity scheme: serials are '<UidPrefix><counter>'.
METHOD Setup : BOOL
VAR_INPUT
    UidPrefix : STRING(40);
END_VAR
IF UidPrefix = '' THEN
    Setup := FALSE;
    RETURN;
END_IF
_prefix := UidPrefix;
_configured := TRUE;
Setup := TRUE;
END_METHOD

// BY_POSITION: the station itself is the identity authority — assign the next
// serial when no Uid is carried yet. FALSE only when unconfigured (§3.16.2:
// the caller faults CARRIER_READ_FAILED; never a silent continue).
METHOD ReadContext : BOOL
VAR_IN_OUT
    Ctx : ST_PartContext;
END_VAR
IF NOT _configured THEN
    ReadContext := FALSE;
    RETURN;
END_IF
IF Ctx.Uid = '' THEN
    _serial := _serial + 1;
    Ctx.Uid := CONCAT(_prefix, UDINT_TO_STRING(_serial));
END_IF
Ctx.Present := TRUE;
Ctx.CarrierKind := E_CarrierKind.BY_POSITION;
ReadContext := TRUE;
END_METHOD

// keep the produced result locally (bounded ring, newest at ProducedHead).
METHOD WriteResult : BOOL
VAR_INPUT
    Ctx : ST_PartContext;
END_VAR
IF NOT _configured THEN
    WriteResult := FALSE;
    RETURN;
END_IF
ProducedHead := ProducedHead + 1;
IF ProducedHead > PL_Fraktal.MAX_RECIPES THEN
    ProducedHead := 1;
END_IF
Produced[ProducedHead] := Ctx.Result;
ProducedUids[ProducedHead] := Ctx.Uid;
WriteResult := TRUE;
END_METHOD

END_FUNCTION_BLOCK

// ---- Connectivity/FB_SimByteChannel.TcPOU
// Core §3.15.1a — scripted in-memory channel: device CMs are TcUnit-tested
// end-to-end with NO socket and NO vendor hardware. Script(Expect, Reply):
// when a sent line matches Expect, Reply is delivered on the next Poll.
FUNCTION_BLOCK FB_SimByteChannel IMPLEMENTS I_ByteChannel
VAR_INPUT
    SwallowNext : BOOL;               // eat the next request (drives timeout tests)
END_VAR
VAR
    _state  : E_ByteChannelState;
    _expect : ARRAY[1..8] OF STRING(255);
    _reply  : ARRAY[1..8] OF STRING(255);
    _n      : INT;
    _pend   : STRING(255);            // reply awaiting delivery
END_VAR

; // driven via Tick/methods

METHOD Script : BOOL
VAR_INPUT
    Expect : STRING(255);
    Reply  : STRING(255);
END_VAR
IF _n >= 8 THEN
    Script := FALSE;
    RETURN;
END_IF
_n := _n + 1;
_expect[_n] := Expect;
_reply[_n] := Reply;
Script := TRUE;
END_METHOD

METHOD Open : BOOL
VAR_INPUT
    Host : STRING(80);
    Port : UINT;
END_VAR
_state := E_ByteChannelState.OPEN;   // sim opens instantly
Open := TRUE;
END_METHOD

METHOD Close : BOOL
_state := E_ByteChannelState.CLOSED;
Close := TRUE;
END_METHOD

METHOD Send : BOOL
VAR_INPUT
    Text : STRING(255);
END_VAR
VAR
    i : INT;
END_VAR
IF _state <> E_ByteChannelState.OPEN THEN
    Send := FALSE;
    RETURN;
END_IF
IF SwallowNext THEN
    SwallowNext := FALSE;             // request eaten: no reply -> caller times out
    Send := TRUE;
    RETURN;
END_IF
FOR i := 1 TO _n DO
    IF _expect[i] = Text THEN
        _pend := _reply[i];
        EXIT;
    END_IF
END_FOR
Send := TRUE;
END_METHOD

METHOD Poll : INT
VAR_IN_OUT
    Buffer : STRING(255);
END_VAR
Poll := 0;
IF _pend <> '' THEN
    Poll := LEN(_pend);
    Buffer := CONCAT(Buffer, _pend);
    _pend := '';
END_IF
END_METHOD

METHOD State : E_ByteChannelState
State := _state;
END_METHOD

METHOD Tick : BOOL
Tick := TRUE;
END_METHOD

END_FUNCTION_BLOCK

// ---- Connectivity/FB_TcpChannelTc3.TcPOU
// [TC3] SKELETON — I_ByteChannel over Tc2_TcpIp (TF6310), TC3 §3.15. Structure and
// building blocks named; bodies are TODO for the integrator, who MUST verify FB
// signatures, the TF6310 license, and the TcpIpServer prerequisite against Beckhoff
// InfoSys for the pinned TwinCAT version. Until implemented, State() = CLOSED.
FUNCTION_BLOCK FB_TcpChannelTc3 IMPLEMENTS I_ByteChannel
VAR
    // Tc2_TcpIp building blocks (uncomment when the library is referenced):
    // _connect : FB_SocketConnect;
    // _close   : FB_SocketClose;
    // _send    : FB_SocketSend;
    // _recv    : FB_SocketReceive;
    _state : E_ByteChannelState;
END_VAR

; // driven via Tick

METHOD Open : BOOL
VAR_INPUT
    Host : STRING(80);
    Port : UINT;
END_VAR
// TODO(integrator): kick _connect(sRemoteHost := Host, nRemotePort := Port, ...);
// _state := OPENING; completion observed in Tick(). Verify param names (InfoSys).
Open := FALSE;   // skeleton
END_METHOD

METHOD Close : BOOL
// TODO(integrator): _close(hSocket := ...); _state := CLOSED;
Close := FALSE;
END_METHOD

METHOD Send : BOOL
VAR_INPUT
    Text : STRING(255);
END_VAR
// TODO(integrator): _send(hSocket := ..., pSrc := ADR(Text), cbLen := LEN(Text));
Send := FALSE;
END_METHOD

METHOD Poll : INT
VAR_IN_OUT
    Buffer : STRING(255);
END_VAR
// TODO(integrator): _recv into a byte buffer, append printable chars to Buffer.
Poll := 0;
END_METHOD

METHOD State : E_ByteChannelState
State := _state;
END_METHOD

METHOD Tick : BOOL
// TODO(integrator): advance _connect/_send/_recv state machines; map completion/
// error onto _state (OPENING -> OPEN on connect done; any bErr -> FAULT).
Tick := TRUE;
END_METHOD

END_FUNCTION_BLOCK

// ---- DeviceCMs/FB_TcpCodeReaderCM.TcPOU
// Core §3.15.1a — CATEGORY CM: triggered TCP/ASCII code reader (barcode/DMC),
// vendor-neutral. Configure for most readers; extend only for special features.
// Optional match-code verification: ParCmd.MatchCode <> ''.
// Publishes: ParCfg, ParCmd, OutCmd, OutImm. Feeds Annex E.
{attribute 'OPC.UA.DA' := '1'}
FUNCTION_BLOCK FB_TcpCodeReaderCM EXTENDS FB_AsciiDeviceCM
VAR_INPUT
    ParCfg : ST_TcpCodeReaderParCfg;
    ParCmd : ST_TcpCodeReaderParCmd;
END_VAR
VAR_OUTPUT
    OutCmd : ST_TcpCodeReaderOutCmd;
    OutImm : ST_TcpCodeReaderOutImm;
END_VAR
VAR
    _done : BOOL;
    _sent : BOOL;
END_VAR

Cyclic();

METHOD Setup : BOOL
VAR_INPUT
    Name : STRING(80);
    Chan : I_ByteChannel;
    DevHost : STRING(80);
    DevPort : UINT;
END_VAR
_M_SetName(Name);
_M_PublishCommand(Value := 1, Label := 'std.command.triggerRead');
ParCfg.Host := DevHost;
ParCfg.Port := DevPort;
Setup := SetupDevice(Chan := Chan, DevHost := DevHost, DevPort := DevPort);
END_METHOD

METHOD PROTECTED _M_Dispatch
IF _manualReq THEN
    _manualReq := FALSE;
    IF _manualCmd = 1 THEN
        _sent := SendRequest(Text := ParCfg.TriggerCmd);
        IF _sent THEN OutCmd.Code := ''; OutCmd.NoRead := FALSE; OutCmd.MatchOk := FALSE; END_IF
    ELSE
        _M_Fault(E_Reason.UNSUPPORTED_COMMAND, 'std.error.unsupportedCodeReaderCommand');
        RETURN;
    END_IF
END_IF
IF Execute THEN
    IF NOT _sent THEN
        _M_TagCommand(Id := 1, Label := 'std.command.triggerRead');
        _sent := SendRequest(Text := ParCfg.TriggerCmd);
        IF _sent THEN
            OutCmd.Code := '';
            OutCmd.NoRead := FALSE;
            OutCmd.MatchOk := FALSE;
        END_IF
    ELSIF _done THEN
        _sent := FALSE;
        _done := FALSE;
        _M_Complete();
    END_IF
ELSE
    _sent := FALSE;
    _done := FALSE;
END_IF
END_METHOD

METHOD PROTECTED OnCyclic : DINT
OnCyclic := SUPER^.OnCyclic();
Host := ParCfg.Host;
Port := ParCfg.Port;
Terminator := ParCfg.Terminator;
RespTimeout := ParCfg.RespTimeout;
OutImm.LinkState := LinkState;
OutImm.LastResponse := LastResponse;
OutImm.Diagnostic := Status.Diagnostic;
END_METHOD

// generic read parse: NoReadText or the decoded symbol; optional match verify.
METHOD PROTECTED _M_OnResponse
VAR_INPUT
    Response : STRING(255);
END_VAR
OutCmd.NoRead := (Response = ParCfg.NoReadText);
IF OutCmd.NoRead THEN OutCmd.Code := ''; END_IF
IF NOT OutCmd.NoRead THEN
    OutCmd.Code := Response;             // -> traceability (Annex E)
END_IF
IF ParCmd.MatchCode <> '' THEN
    OutCmd.MatchOk := (NOT OutCmd.NoRead) AND (Response = ParCmd.MatchCode);
ELSE
    OutCmd.MatchOk := NOT OutCmd.NoRead;
END_IF
_done := TRUE;
END_METHOD

METHOD PROTECTED _M_PublishStatus
SUPER^._M_PublishStatus();
OutImm.Diagnostic := Status.Diagnostic;
END_METHOD

END_FUNCTION_BLOCK

// ---- DeviceCMs/FB_TcpVisionCM.TcPOU
// Core §3.15.1a — CATEGORY CM: triggered TCP/ASCII vision system, vendor-neutral.
// Configure for most devices (protocol strings below, §3.8-able, VERIFY vs the
// vendor manual); extend only for genuinely special features. Function over
// vendor: the forest shows 'vision inspection', never a brand.
// Publishes: ParCfg, ParCmd, OutCmd, OutImm.
{attribute 'OPC.UA.DA' := '1'}
FUNCTION_BLOCK FB_TcpVisionCM EXTENDS FB_AsciiDeviceCM
VAR_INPUT
    ParCfg : ST_TcpVisionParCfg;
    ParCmd : ST_TcpVisionParCmd;
END_VAR
VAR_OUTPUT
    OutCmd : ST_TcpVisionOutCmd;
    OutImm : ST_TcpVisionOutImm;
END_VAR
VAR
    _done : BOOL;
    _sent : BOOL;
END_VAR

Cyclic();

// wire name + transport + endpoint; publishes the manual Trigger command (§7.6.1)
METHOD Setup : BOOL
VAR_INPUT
    Name : STRING(80);
    Chan : I_ByteChannel;
    DevHost : STRING(80);
    DevPort : UINT;
END_VAR
_M_SetName(Name);
_M_PublishCommand(Value := 1, Label := 'std.command.trigger');
ParCfg.Host := DevHost;
ParCfg.Port := DevPort;
Setup := SetupDevice(Chan := Chan, DevHost := DevHost, DevPort := DevPort);
END_METHOD

METHOD PROTECTED _M_Dispatch
IF _manualReq THEN
    _manualReq := FALSE;
    IF _manualCmd = 1 THEN
        _sent := SendRequest(Text := ParCfg.TriggerCmd); // §7.6.1: one request through normal dispatch
        IF _sent THEN OutCmd.JudgeOk := FALSE; OutCmd.ResultData := ''; END_IF
    ELSE
        _M_Fault(E_Reason.UNSUPPORTED_COMMAND, 'std.error.unsupportedVisionCommand');
        RETURN;
    END_IF
END_IF
IF Execute THEN
    IF NOT _sent THEN
        _M_TagCommand(Id := 1, Label := 'std.command.inspect');
        _sent := SendRequest(Text := ParCfg.TriggerCmd);
        IF _sent THEN
            OutCmd.JudgeOk := FALSE;
            OutCmd.ResultData := '';
        END_IF
    ELSIF _done THEN
        _sent := FALSE;
        _done := FALSE;
        _M_Complete();
    END_IF
ELSE
    _sent := FALSE;
    _done := FALSE;
END_IF
END_METHOD

// generic judgement parse: OkPrefix/NgPrefix + optional payload after ResultSep.
// Devices with special result formats override THIS, nothing else.
METHOD PROTECTED _M_OnResponse
VAR_INPUT
    Response : STRING(255);
END_VAR
VAR
    pLen : INT;
END_VAR
IF LEFT(Response, LEN(ParCfg.OkPrefix)) = ParCfg.OkPrefix THEN
    OutCmd.JudgeOk := TRUE;
    pLen := LEN(ParCfg.OkPrefix);
ELSIF LEFT(Response, LEN(ParCfg.NgPrefix)) = ParCfg.NgPrefix THEN
    OutCmd.JudgeOk := FALSE;
    pLen := LEN(ParCfg.NgPrefix);
ELSE
    _M_FaultN(PL_TcpDevReasons.DEV_PROTOCOL, 'std.error.unexpectedVisionReply');
    RETURN;
END_IF
OutCmd.ResultData := '';
IF LEN(Response) > pLen + LEN(ParCfg.ResultSep) THEN
    IF MID(Response, LEN(ParCfg.ResultSep), pLen + 1) = ParCfg.ResultSep THEN
        OutCmd.ResultData := RIGHT(Response, LEN(Response) - pLen - LEN(ParCfg.ResultSep));
    END_IF
END_IF
_done := TRUE;
END_METHOD

METHOD PROTECTED OnCyclic : DINT
OnCyclic := SUPER^.OnCyclic();
Host := ParCfg.Host;
Port := ParCfg.Port;
Terminator := ParCfg.Terminator;
RespTimeout := ParCfg.RespTimeout;
OutImm.LinkState := LinkState;
OutImm.LastResponse := LastResponse;
OutImm.Diagnostic := Status.Diagnostic;
END_METHOD

METHOD PROTECTED _M_PublishStatus
SUPER^._M_PublishStatus();
OutImm.Diagnostic := Status.Diagnostic;
END_METHOD

END_FUNCTION_BLOCK

// ---- PermIntlk/FB_PermIntlk.TcPOU
// Core §7.2 — the standard permissive/interlock container: fixed container,
// author-chosen condition language (LD/ST/FBD drive Cond[i], TRUE = OK).
// First FALSE, non-bypassed, defined condition is the first-out reason (Core §6.9).
FUNCTION_BLOCK FB_PermIntlk
VAR_INPUT
    Cond : ARRAY[1..PL_Fraktal.MAX_PERMINTLK_COND] OF BOOL;   // author drives these (TRUE = OK)
END_VAR
VAR_OUTPUT
    AllOk       : BOOL;   // every defined, non-bypassed condition is TRUE
    AnyBypassed : BOOL;   // at least one defined condition is bypassed
    FirstFailed : INT;    // lowest index of a FALSE, non-bypassed condition; 0 = none
END_VAR
VAR
    _conds   : ARRAY[1..PL_Fraktal.MAX_PERMINTLK_COND] OF ST_IntlkCond;
    _bypass  : ARRAY[1..PL_Fraktal.MAX_PERMINTLK_COND] OF BOOL;
    _diag    : ST_Diagnostic;
    _lastFf  : INT;
END_VAR
VAR
    i   : INT;
    ok  : BOOL;
    byp : BOOL;
    ff  : INT;
END_VAR

// evaluate every defined condition; first FALSE (non-bypassed) is the first-out
ok := TRUE;
byp := FALSE;
ff := 0;
FOR i := 1 TO PL_Fraktal.MAX_PERMINTLK_COND DO
    IF _conds[i].Defined THEN
        IF _bypass[i] THEN
            byp := TRUE;                       // bypassed => not evaluated, but flagged (Core §7.3)
        ELSIF NOT Cond[i] THEN
            ok := FALSE;
            IF ff = 0 THEN
                ff := i;
            END_IF
        END_IF
    END_IF
END_FOR
AllOk       := ok;
AnyBypassed := byp;
FirstFailed := ff;

IF ff = 0 THEN
    _diag.ReasonCode  := E_Reason.NONE;
    _diag.Description := '';
ELSE
    IF ff <> _lastFf THEN
        _diag.Since := F_Now();                // stamp only on a NEW first-out (Core §8.8)
    END_IF
    _diag.ReasonCode  := _conds[ff].Reason;
    _diag.Description := _conds[ff].Description;
    _diag.Severity    := E_Severity.LOW;       // pending reason while blocked; owner promotes on fault
    _diag.Category    := E_Category.PROCESS;
    // SourcePath is set by the OWNER when copying the diagnostic up (Core §7.2 usage contract)
END_IF
_lastFf := ff;

// Core §7.2 — clears all bypasses
METHOD ClearBypass : BOOL
VAR
    i : INT;
END_VAR
FOR i := 1 TO PL_Fraktal.MAX_PERMINTLK_COND DO
    _bypass[i] := FALSE;
END_FOR
ClearBypass := TRUE;
END_METHOD

// Core §7.2 — declare one condition record (typically once, in the owner's Setup/init).
// Bounds-checked per Core §5.6: an out-of-range index is rejected, never written.
METHOD Define : BOOL
VAR_INPUT
    Index       : INT;
    Description : STRING(255);
    Reason      : E_Reason;
    Bypassable  : BOOL;
END_VAR
IF (Index < 1) OR (Index > PL_Fraktal.MAX_PERMINTLK_COND) THEN
    Define := FALSE;
    RETURN;
END_IF
_conds[Index].Defined     := TRUE;
_conds[Index].Description := Description;
_conds[Index].Reason      := Reason;
_conds[Index].Bypassable  := Bypassable;
Define := TRUE;
END_METHOD

// Core §7.2/§7.3 — succeeds only for a defined, explicitly-bypassable condition
METHOD SetBypass : BOOL
VAR_INPUT
    Index : INT;
    On    : BOOL;
END_VAR
IF (Index < 1) OR (Index > PL_Fraktal.MAX_PERMINTLK_COND) THEN
    SetBypass := FALSE;
    RETURN;
END_IF
IF _conds[Index].Defined AND _conds[Index].Bypassable THEN
    _bypass[Index] := On;
    SetBypass := TRUE;
ELSE
    SetBypass := FALSE;
END_IF
END_METHOD

// Core §7.2 — first-out: Reason + Description of FirstFailed (ReasonCode = NONE when AllOk)
PROPERTY Diagnostic : ST_Diagnostic
GET
Diagnostic := _diag;
END_GET
END_PROPERTY

// Core §7.8 — append EVERY currently-failed (defined, non-bypassed, FALSE) condition
// to a release report as INTERLOCK reasons. Returns the new count. Complete list,
// not just first-out. Pure query: never commands, never mutates conditions.
METHOD AppendFailed : INT
VAR_INPUT
    SourcePath : STRING(255);   // owner supplied explicitly; the container is reusable
END_VAR
VAR_IN_OUT
    Report : ST_ReleaseReport;
END_VAR
VAR
    i : INT;
END_VAR
FOR i := 1 TO PL_Fraktal.MAX_PERMINTLK_COND DO
    IF _conds[i].Defined AND NOT _bypass[i] AND NOT Cond[i] THEN
        IF Report.Count < PL_Fraktal.MAX_RELEASE_REASONS THEN
            Report.Count := Report.Count + 1;
            Report.Reasons[Report.Count].Description := _conds[i].Description;
            Report.Reasons[Report.Count].ReasonCode  := _conds[i].Reason;
            Report.Reasons[Report.Count].SourcePath  := SourcePath;
            Report.Reasons[Report.Count].Kind        := E_ReleaseKind.INTERLOCK;
            Report.Reasons[Report.Count].Bypassable  := _conds[i].Bypassable;
        END_IF
    END_IF
END_FOR
AppendFailed := Report.Count;
END_METHOD

END_FUNCTION_BLOCK
